LIN {X 0,Y 466.726,Z 1100.087,A -85,B 0,C 180,E1 19216.382,E2 19216.382} C_VEL
LIN {X 0,Y 459.016,Z 1120.699,A -85,B 0,C 180,E1 19214.007,E2 19214.007} C_VEL
LIN {X 0,Y 452.977,Z 1136.346,A -85,B 0,C 180,E1 19211.936,E2 19211.936} C_VEL
LIN {X 0,Y 447.551,Z 1150.209,A -85,B 0,C 180,E1 19209.871,E2 19209.871} C_VEL
LIN {X 0,Y 442.276,Z 1163.7,A -85,B 0,C 180,E1 19207.609,E2 19207.609} C_VEL
LIN {X 0,Y 436.923,Z 1177.533,A -85,B 0,C 180,E1 19204.987,E2 19204.987} C_VEL
LIN {X 0,Y 430.904,Z 1193.503,A -85,B 0,C 180,E1 19201.464,E2 19201.464} C_VEL
LIN {X 0,Y 426.882,Z 1204.833,A -85,B 0,C 180,E1 19198.535,E2 19198.535} C_VEL
LIN {X 0,Y 423.763,Z 1214.343,A -85,B 0,C 180,E1 19195.723,E2 19195.723} C_VEL
LIN {X 0,Y 421.063,Z 1223.466,A -85,B 0,C 180,E1 19192.617,E2 19192.617} C_VEL
LIN {X 0,Y 418.595,Z 1233.141,A -85,B 0,C 180,E1 19188.66,E2 19188.66} C_VEL
LIN {X 0,Y 417.349,Z 1239.293,A -85,B 0,C 180,E1 19185.558,E2 19185.558} C_VEL
LIN {X 0,Y 416.602,Z 1244.084,A -85,B 0,C 180,E1 19182.608,E2 19182.608} C_VEL
LIN {X 0,Y 416.536,Z 1244.656,A -85,B 0,C 180,E1 19182.208,E2 19182.208} C_VEL
LIN {X 0,Y 415.382,Z 1246.217,A -85,B 0,C 180,E1 19181.171,E2 19181.171} C_VEL
LIN {X 0,Y 408.591,Z 1249.799,A -85,B 0,C 180,E1 19178.242,E2 19178.242} C_VEL
LIN {X 0,Y 408.036,Z 1250.419,A -85,B 0,C 180,E1 19177.468,E2 19177.468} C_VEL
LIN {X 0,Y 407.953,Z 1252.387,A -85,B 0,C 180,E1 19174.492,E2 19174.492} C_VEL
LIN {X 0,Y 407.933,Z 1253.358,A -85,B 0,C 180,E1 19171.679,E2 19171.679} C_VEL
LIN {X 0,Y 407.906,Z 1253.459,A -85,B 0,C 180,E1 19168.87,E2 19168.87} C_VEL
LIN {X 0,Y 407.952,Z 1252.658,A -85,B 0,C 180,E1 19165.999,E2 19165.999} C_VEL
LIN {X 0,Y 408.019,Z 1250.929,A -85,B 0,C 180,E1 19163.097,E2 19163.097} C_VEL
LIN {X 0,Y 408.169,Z 1248.351,A -85,B 0,C 180,E1 19160.263,E2 19160.263} C_VEL
LIN {X 0,Y 408.603,Z 1244.86,A -85,B 0,C 180,E1 19157.415,E2 19157.415} C_VEL
LIN {X 0,Y 409.295,Z 1240.436,A -85,B 0,C 180,E1 19154.551,E2 19154.551} C_VEL
LIN {X 0,Y 410.489,Z 1234.748,A -85,B 0,C 180,E1 19151.533,E2 19151.533} C_VEL
LIN {X 0,Y 412.211,Z 1227.955,A -85,B 0,C 180,E1 19148.508,E2 19148.508} C_VEL
LIN {X 0,Y 415.091,Z 1218.417,A -85,B 0,C 180,E1 19144.91,E2 19144.91} C_VEL
LIN {X 0,Y 418.953,Z 1206.868,A -85,B 0,C 180,E1 19141.328,E2 19141.328} C_VEL
LIN {X 0,Y 422.851,Z 1196.299,A -85,B 0,C 180,E1 19138.489,E2 19138.489} C_VEL
LIN {X 0,Y 427.224,Z 1185.009,A -85,B 0,C 180,E1 19135.821,E2 19135.821} C_VEL
LIN {X 0,Y 433.187,Z 1170.311,A -85,B 0,C 180,E1 19132.782,E2 19132.782} C_VEL
LIN {X 0,Y 440.181,Z 1153.04,A -85,B 0,C 180,E1 19129.751,E2 19129.751} C_VEL
LIN {X 0,Y 446.161,Z 1138.346,A -85,B 0,C 180,E1 19127.504,E2 19127.504} C_VEL
LIN {X 0,Y 452.131,Z 1123.44,A -85,B 0,C 180,E1 19125.484,E2 19125.484} C_VEL
LIN {X 0,Y 458.329,Z 1107.59,A -85,B 0,C 180,E1 19123.582,E2 19123.582} C_VEL
LIN {X 0,Y 466.092,Z 1087.076,A -85,B 0,C 180,E1 19121.425,E2 19121.425} C_VEL
LIN {X 0,Y 473.649,Z 1065.436,A -85,B 0,C 180,E1 19119.499,E2 19119.499} C_VEL
LIN {X 0,Y 479.534,Z 1047.568,A -85,B 0,C 180,E1 19118.112,E2 19118.112} C_VEL
LIN {X 0,Y 485.331,Z 1028.607,A -85,B 0,C 180,E1 19116.819,E2 19116.819} C_VEL
LIN {X 0,Y 491.208,Z 1007.732,A -85,B 0,C 180,E1 19115.585,E2 19115.585} C_VEL
LIN {X 0,Y 497.603,Z 982.362,A -85,B 0,C 180,E1 19114.319,E2 19114.319} C_VEL
LIN {X 0,Y 502.722,Z 958.44,A -85,B 0,C 180,E1 19113.342,E2 19113.342} C_VEL
LIN {X 0,Y 506.626,Z 937.283,A -85,B 0,C 180,E1 19112.624,E2 19112.624} C_VEL
LIN {X 0,Y 509.947,Z 915.923,A -85,B 0,C 180,E1 19112.03,E2 19112.03} C_VEL
LIN {X 0,Y 512.846,Z 892.593,A -85,B 0,C 180,E1 19111.515,E2 19111.515} C_VEL
LIN {X 0,Y 515.629,Z 856.761,A -85,B 0,C 180,E1 19110.915,E2 19110.915} C_VEL
LIN {X 0,Y 529.358,Z 635.561,A -85,B 0,C 180,E1 19107.486,E2 19107.486} C_VEL
LIN {X 0,Y 533.456,Z 570.989,A -85,B 0,C 180,E1 19106.464,E2 19106.464} C_VEL
LIN {X 0,Y 524.737,Z 558.021,A -85,B 0,C 180,E1 19104.036,E2 19104.036} C_VEL
LIN {X 0,Y 516.788,Z 546.823,A -85,B 0,C 180,E1 19101.539,E2 19101.539} C_VEL
LIN {X 0,Y 510.867,Z 538.783,A -85,B 0,C 180,E1 19099.435,E2 19099.435} C_VEL
LIN {X 0,Y 506.895,Z 533.497,A -85,B 0,C 180,E1 19097.863,E2 19097.863} C_VEL
LIN {X 0,Y 503.376,Z 528.832,A -85,B 0,C 180,E1 19096.324,E2 19096.324} C_VEL
LIN {X 0,Y 499.419,Z 523.648,A -85,B 0,C 180,E1 19094.375,E2 19094.375} C_VEL
LIN {X 0,Y 496.052,Z 519.314,A -85,B 0,C 180,E1 19092.455,E2 19092.455} C_VEL
LIN {X 0,Y 495.152,Z 518.176,A -85,B 0,C 180,E1 19091.887,E2 19091.887} C_VEL
LIN {X 0,Y 491.947,Z 514.441,A -85,B 0,C 180,E1 19089.594,E2 19089.594} C_VEL
LIN {X 0,Y 490.94,Z 512.514,A -85,B 0,C 180,E1 19088.668,E2 19088.668} C_VEL
LIN {X 0,Y 487.515,Z 509.124,A -85,B 0,C 180,E1 19084.706,E2 19084.706} C_VEL
LIN {X 0,Y 486.689,Z 506.403,A -85,B 0,C 180,E1 19082.355,E2 19082.355} C_VEL
LIN {X 0,Y 486.775,Z 506.534,A -85,B 0,C 180,E1 19077.763,E2 19077.763} C_VEL
LIN {X 0,Y 488.567,Z 510.725,A -85,B 0,C 180,E1 19074.127,E2 19074.127} C_VEL
LIN {X 0,Y 491.202,Z 512.848,A -85,B 0,C 180,E1 19071.513,E2 19071.513} C_VEL
LIN {X 0,Y 493.665,Z 516.868,A -85,B 0,C 180,E1 19069.497,E2 19069.497} C_VEL
LIN {X 0,Y 495.884,Z 519.004,A -85,B 0,C 180,E1 19068.072,E2 19068.072} C_VEL
LIN {X 0,Y 499.313,Z 523.558,A -85,B 0,C 180,E1 19066.095,E2 19066.095} C_VEL
LIN {X 0,Y 500.82,Z 525.628,A -85,B 0,C 180,E1 19065.312,E2 19065.312} C_VEL
LIN {X 0,Y 505.099,Z 531.129,A -85,B 0,C 180,E1 19063.319,E2 19063.319} C_VEL
LIN {X 0,Y 511.053,Z 540.056,A -85,B 0,C 180,E1 19060.87,E2 19060.87} C_VEL
LIN {X 0,Y 516.454,Z 548.16,A -85,B 0,C 180,E1 19058.923,E2 19058.923} C_VEL
LIN {X 0,Y 524.596,Z 561.043,A -85,B 0,C 180,E1 19056.316,E2 19056.316} C_VEL
LIN {X 0,Y 533.578,Z 575.978,A -85,B 0,C 180,E1 19053.779,E2 19053.779} C_VEL
LIN {X 0,Y 520.443,Z 784.729,A -85,B 0,C 180,E1 19050.532,E2 19050.532} C_VEL
LIN {X 0,Y 513.397,Z 898.299,A -85,B 0,C 180,E1 19048.753,E2 19048.753} C_VEL
LIN {X 0,Y 510.438,Z 925.967,A -85,B 0,C 180,E1 19048.226,E2 19048.226} C_VEL
LIN {X 0,Y 506.32,Z 952.366,A -85,B 0,C 180,E1 19047.555,E2 19047.555} C_VEL
LIN {X 0,Y 502.372,Z 973.666,A -85,B 0,C 180,E1 19046.874,E2 19046.874} C_VEL
LIN {X 0,Y 497.981,Z 994.234,A -85,B 0,C 180,E1 19046.088,E2 19046.088} C_VEL
LIN {X 0,Y 492.921,Z 1015.345,A -85,B 0,C 180,E1 19045.132,E2 19045.132} C_VEL
LIN {X 0,Y 486.06,Z 1040.963,A -85,B 0,C 180,E1 19043.75,E2 19043.75} C_VEL
LIN {X 0,Y 479.409,Z 1062.995,A -85,B 0,C 180,E1 19042.331,E2 19042.331} C_VEL
LIN {X 0,Y 473.078,Z 1082.578,A -85,B 0,C 180,E1 19040.872,E2 19040.872} C_VEL
LIN {X 0,Y 466.468,Z 1101.878,A -85,B 0,C 180,E1 19039.224,E2 19039.224} C_VEL
LIN {X 0,Y 458.48,Z 1124.086,A -85,B 0,C 180,E1 19037.033,E2 19037.033} C_VEL
LIN {X 0,Y 450.994,Z 1143.777,A -85,B 0,C 180,E1 19034.747,E2 19034.747} C_VEL
LIN {X 0,Y 445.06,Z 1159.134,A -85,B 0,C 180,E1 19032.722,E2 19032.722} C_VEL
LIN {X 0,Y 439.157,Z 1174.316,A -85,B 0,C 180,E1 19030.464,E2 19030.464} C_VEL
LIN {X 0,Y 432.558,Z 1191.551,A -85,B 0,C 180,E1 19027.545,E2 19027.545} C_VEL
LIN {X 0,Y 426.449,Z 1207.49,A -85,B 0,C 180,E1 19024.378,E2 19024.378} C_VEL
LIN {X 0,Y 421.982,Z 1219.772,A -85,B 0,C 180,E1 19021.583,E2 19021.583} C_VEL
LIN {X 0,Y 418.242,Z 1230.826,A -85,B 0,C 180,E1 19018.725,E2 19018.725} C_VEL
LIN {X 0,Y 414.529,Z 1242.95,A -85,B 0,C 180,E1 19015.126,E2 19015.126} C_VEL
LIN {X 0,Y 411.805,Z 1253.015,A -85,B 0,C 180,E1 19011.514,E2 19011.514} C_VEL
LIN {X 0,Y 410.172,Z 1260.206,A -85,B 0,C 180,E1 19008.481,E2 19008.481} C_VEL
LIN {X 0,Y 409.136,Z 1265.988,A -85,B 0,C 180,E1 19005.6,E2 19005.6} C_VEL
LIN {X 0,Y 408.459,Z 1270.971,A -85,B 0,C 180,E1 19002.59,E2 19002.59} C_VEL
LIN {X 0,Y 408.085,Z 1274.707,A -85,B 0,C 180,E1 18999.739,E2 18999.739} C_VEL
LIN {X 0,Y 407.978,Z 1277.483,A -85,B 0,C 180,E1 18996.903,E2 18996.903} C_VEL
LIN {X 0,Y 407.935,Z 1279.311,A -85,B 0,C 180,E1 18994.082,E2 18994.082} C_VEL
LIN {X 0,Y 407.921,Z 1280.177,A -85,B 0,C 180,E1 18991.411,E2 18991.411} C_VEL
LIN {X 0,Y 407.915,Z 1280.202,A -85,B 0,C 180,E1 18988.742,E2 18988.742} C_VEL
LIN {X 0,Y 407.935,Z 1279.368,A -85,B 0,C 180,E1 18986.032,E2 18986.032} C_VEL
LIN {X 0,Y 407.973,Z 1277.61,A -85,B 0,C 180,E1 18983.251,E2 18983.251} C_VEL
LIN {X 0,Y 408.073,Z 1274.886,A -85,B 0,C 180,E1 18980.416,E2 18980.416} C_VEL
LIN {X 0,Y 408.435,Z 1271.203,A -85,B 0,C 180,E1 18977.566,E2 18977.566} C_VEL
LIN {X 0,Y 409.082,Z 1266.273,A -85,B 0,C 180,E1 18974.556,E2 18974.556} C_VEL
LIN {X 0,Y 410.105,Z 1260.544,A -85,B 0,C 180,E1 18971.676,E2 18971.676} C_VEL
LIN {X 0,Y 411.701,Z 1253.406,A -85,B 0,C 180,E1 18968.644,E2 18968.644} C_VEL
LIN {X 0,Y 414.263,Z 1243.805,A -85,B 0,C 180,E1 18965.168,E2 18965.168} C_VEL
LIN {X 0,Y 418.052,Z 1231.399,A -85,B 0,C 180,E1 18961.431,E2 18961.431} C_VEL
LIN {X 0,Y 421.762,Z 1220.406,A -85,B 0,C 180,E1 18958.572,E2 18958.572} C_VEL
LIN {X 0,Y 425.986,Z 1208.695,A -85,B 0,C 180,E1 18955.885,E2 18955.885} C_VEL
LIN {X 0,Y 431.201,Z 1194.919,A -85,B 0,C 180,E1 18953.099,E2 18953.099} C_VEL
LIN {X 0,Y 438.495,Z 1176.02,A -85,B 0,C 180,E1 18949.809,E2 18949.809} C_VEL
LIN {X 0,Y 444.678,Z 1160.077,A -85,B 0,C 180,E1 18947.416,E2 18947.416} C_VEL
LIN {X 0,Y 450.753,Z 1144.339,A -85,B 0,C 180,E1 18945.328,E2 18945.328} C_VEL
LIN {X 0,Y 457.565,Z 1126.379,A -85,B 0,C 180,E1 18943.228,E2 18943.228} C_VEL
LIN {X 0,Y 466.103,Z 1102.816,A -85,B 0,C 180,E1 18940.866,E2 18940.866} C_VEL
LIN {X 0,Y 472.749,Z 1083.429,A -85,B 0,C 180,E1 18939.202,E2 18939.202} C_VEL
LIN {X 0,Y 478.837,Z 1064.661,A -85,B 0,C 180,E1 18937.793,E2 18937.793} C_VEL
LIN {X 0,Y 484.915,Z 1044.638,A -85,B 0,C 180,E1 18936.483,E2 18936.483} C_VEL
LIN {X 0,Y 491.767,Z 1019.829,A -85,B 0,C 180,E1 18935.09,E2 18935.09} C_VEL
LIN {X 0,Y 497.452,Z 996.33,A -85,B 0,C 180,E1 18934.005,E2 18934.005} C_VEL
LIN {X 0,Y 502.002,Z 975.19,A -85,B 0,C 180,E1 18933.184,E2 18933.184} C_VEL
LIN {X 0,Y 505.927,Z 954.249,A -85,B 0,C 180,E1 18932.506,E2 18932.506} C_VEL
LIN {X 0,Y 509.434,Z 932.151,A -85,B 0,C 180,E1 18931.924,E2 18931.924} C_VEL
LIN {X 0,Y 512.865,Z 904.139,A -85,B 0,C 180,E1 18931.35,E2 18931.35} C_VEL
LIN {X 0,Y 515.951,Z 857.879,A -85,B 0,C 180,E1 18930.607,E2 18930.607} C_VEL
LIN {X 0,Y 529.334,Z 640.596,A -85,B 0,C 180,E1 18927.234,E2 18927.234} C_VEL
LIN {X 0,Y 533.472,Z 575.938,A -85,B 0,C 180,E1 18926.223,E2 18926.223} C_VEL
LIN {X 0,Y 524.4,Z 560.859,A -85,B 0,C 180,E1 18923.664,E2 18923.664} C_VEL
LIN {X 0,Y 516.019,Z 547.617,A -85,B 0,C 180,E1 18920.977,E2 18920.977} C_VEL
LIN {X 0,Y 509.259,Z 537.343,A -85,B 0,C 180,E1 18918.487,E2 18918.487} C_VEL
LIN {X 0,Y 503.589,Z 529.163,A -85,B 0,C 180,E1 18916.08,E2 18916.08} C_VEL
LIN {X 0,Y 499.246,Z 523.57,A -85,B 0,C 180,E1 18913.966,E2 18913.966} C_VEL
LIN {X 0,Y 495.613,Z 518.693,A -85,B 0,C 180,E1 18911.875,E2 18911.875} C_VEL
LIN {X 0,Y 492.093,Z 514.875,A -85,B 0,C 180,E1 18909.473,E2 18909.473} C_VEL
LIN {X 0,Y 490.793,Z 512.489,A -85,B 0,C 180,E1 18908.317,E2 18908.317} C_VEL
LIN {X 0,Y 487.383,Z 509.118,A -85,B 0,C 180,E1 18904.471,E2 18904.471} C_VEL
LIN {X 0,Y 486.52,Z 506.4,A -85,B 0,C 180,E1 18902.238,E2 18902.238} C_VEL
LIN {X 0,Y 486.665,Z 506.642,A -85,B 0,C 180,E1 18896.82,E2 18896.82} C_VEL
LIN {X 0,Y 487.967,Z 510.023,A -85,B 0,C 180,E1 18894.119,E2 18894.119} C_VEL
LIN {X 0,Y 491.082,Z 512.857,A -85,B 0,C 180,E1 18890.921,E2 18890.921} C_VEL
LIN {X 0,Y 493.424,Z 516.662,A -85,B 0,C 180,E1 18889.019,E2 18889.019} C_VEL
LIN {X 0,Y 495.739,Z 518.901,A -85,B 0,C 180,E1 18887.537,E2 18887.537} C_VEL
LIN {X 0,Y 499.073,Z 523.419,A -85,B 0,C 180,E1 18885.615,E2 18885.615} C_VEL
LIN {X 0,Y 500.379,Z 525.041,A -85,B 0,C 180,E1 18884.943,E2 18884.943} C_VEL
LIN {X 0,Y 504.758,Z 530.701,A -85,B 0,C 180,E1 18882.892,E2 18882.892} C_VEL
LIN {X 0,Y 508.971,Z 536.338,A -85,B 0,C 180,E1 18881.145,E2 18881.145} C_VEL
LIN {X 0,Y 513.583,Z 542.55,A -85,B 0,C 180,E1 18879.426,E2 18879.426} C_VEL
LIN {X 0,Y 519.796,Z 551.145,A -85,B 0,C 180,E1 18877.343,E2 18877.343} C_VEL
LIN {X 0,Y 526.736,Z 561.091,A -85,B 0,C 180,E1 18875.255,E2 18875.255} C_VEL
LIN {X 0,Y 533.433,Z 571.162,A -85,B 0,C 180,E1 18873.42,E2 18873.42} C_VEL
LIN {X 0,Y 519.648,Z 789.072,A -85,B 0,C 180,E1 18870.039,E2 18870.039} C_VEL
LIN {X 0,Y 513.854,Z 881.148,A -85,B 0,C 180,E1 18868.594,E2 18868.594} C_VEL
LIN {X 0,Y 510.941,Z 908.605,A -85,B 0,C 180,E1 18868.056,E2 18868.056} C_VEL
LIN {X 0,Y 507.028,Z 934.536,A -85,B 0,C 180,E1 18867.364,E2 18867.364} C_VEL
LIN {X 0,Y 503.185,Z 955.72,A -85,B 0,C 180,E1 18866.662,E2 18866.662} C_VEL
LIN {X 0,Y 498.898,Z 976.164,A -85,B 0,C 180,E1 18865.852,E2 18865.852} C_VEL
LIN {X 0,Y 493.586,Z 998.455,A -85,B 0,C 180,E1 18864.811,E2 18864.811} C_VEL
LIN {X 0,Y 486.295,Z 1025.23,A -85,B 0,C 180,E1 18863.298,E2 18863.298} C_VEL
LIN {X 0,Y 480.324,Z 1044.924,A -85,B 0,C 180,E1 18861.982,E2 18861.982} C_VEL
LIN {X 0,Y 474.546,Z 1062.594,A -85,B 0,C 180,E1 18860.637,E2 18860.637} C_VEL
LIN {X 0,Y 468.3,Z 1080.543,A -85,B 0,C 180,E1 18859.087,E2 18859.087} C_VEL
LIN {X 0,Y 461.069,Z 1100.356,A -85,B 0,C 180,E1 18857.126,E2 18857.126} C_VEL
LIN {X 0,Y 452.98,Z 1121.24,A -85,B 0,C 180,E1 18854.702,E2 18854.702} C_VEL
LIN {X 0,Y 446.89,Z 1136.46,A -85,B 0,C 180,E1 18852.672,E2 18852.672} C_VEL
LIN {X 0,Y 441.191,Z 1150.486,A -85,B 0,C 180,E1 18850.564,E2 18850.564} C_VEL
LIN {X 0,Y 435.693,Z 1163.977,A -85,B 0,C 180,E1 18848.279,E2 18848.279} C_VEL
LIN {X 0,Y 430.208,Z 1177.547,A -85,B 0,C 180,E1 18845.678,E2 18845.678} C_VEL
LIN {X 0,Y 423.945,Z 1193.42,A -85,B 0,C 180,E1 18842.143,E2 18842.143} C_VEL
LIN {X 0,Y 419.776,Z 1204.605,A -85,B 0,C 180,E1 18839.22,E2 18839.22} C_VEL
LIN {X 0,Y 416.446,Z 1214.17,A -85,B 0,C 180,E1 18836.363,E2 18836.363} C_VEL
LIN {X 0,Y 413.649,Z 1222.95,A -85,B 0,C 180,E1 18833.347,E2 18833.347} C_VEL
LIN {X 0,Y 411.21,Z 1231.897,A -85,B 0,C 180,E1 18829.746,E2 18829.746} C_VEL
LIN {X 0,Y 409.539,Z 1239.316,A -85,B 0,C 180,E1 18826.007,E2 18826.007} C_VEL
LIN {X 0,Y 408.666,Z 1244.352,A -85,B 0,C 180,E1 18822.857,E2 18822.857} C_VEL
LIN {X 0,Y 408.212,Z 1247.956,A -85,B 0,C 180,E1 18820.008,E2 18820.008} C_VEL
LIN {X 0,Y 408.036,Z 1250.419,A -85,B 0,C 180,E1 18817.468,E2 18817.468} C_VEL
LIN {X 0,Y 407.031,Z 1251.303,A -85,B 0,C 180,E1 18816.394,E2 18816.394} C_VEL
LIN {X 0,Y 402.53,Z 1252.744,A -85,B 0,C 180,E1 18814.442,E2 18814.442} C_VEL
LIN {X 0,Y 400.152,Z 1253.388,A -85,B 0,C 180,E1 18813.044,E2 18813.044} C_VEL
LIN {X 0,Y 399.942,Z 1253.493,A -85,B 0,C 180,E1 18812.565,E2 18812.565} C_VEL
LIN {X 0,Y 399.899,Z 1253.766,A -85,B 0,C 180,E1 18809.134,E2 18809.134} C_VEL
LIN {X 0,Y 399.956,Z 1253.015,A -85,B 0,C 180,E1 18806.123,E2 18806.123} C_VEL
LIN {X 0,Y 400.027,Z 1251.303,A -85,B 0,C 180,E1 18803.103,E2 18803.103} C_VEL
LIN {X 0,Y 400.187,Z 1248.77,A -85,B 0,C 180,E1 18800.212,E2 18800.212} C_VEL
LIN {X 0,Y 400.639,Z 1245.326,A -85,B 0,C 180,E1 18797.307,E2 18797.307} C_VEL
LIN {X 0,Y 401.428,Z 1240.703,A -85,B 0,C 180,E1 18794.241,E2 18794.241} C_VEL
LIN {X 0,Y 402.693,Z 1235.017,A -85,B 0,C 180,E1 18791.163,E2 18791.163} C_VEL
LIN {X 0,Y 404.669,Z 1227.823,A -85,B 0,C 180,E1 18787.909,E2 18787.909} C_VEL
LIN {X 0,Y 408.024,Z 1217.356,A -85,B 0,C 180,E1 18783.977,E2 18783.977} C_VEL
LIN {X 0,Y 411.858,Z 1206.636,A -85,B 0,C 180,E1 18780.627,E2 18780.627} C_VEL
LIN {X 0,Y 415.966,Z 1196.01,A -85,B 0,C 180,E1 18777.743,E2 18777.743} C_VEL
LIN {X 0,Y 420.869,Z 1184.036,A -85,B 0,C 180,E1 18774.9,E2 18774.9} C_VEL
LIN {X 0,Y 428.108,Z 1166.888,A -85,B 0,C 180,E1 18771.415,E2 18771.415} C_VEL
LIN {X 0,Y 434.058,Z 1152.818,A -85,B 0,C 180,E1 18768.96,E2 18768.96} C_VEL
LIN {X 0,Y 440.286,Z 1138.072,A -85,B 0,C 180,E1 18766.693,E2 18766.693} C_VEL
LIN {X 0,Y 446.663,Z 1122.709,A -85,B 0,C 180,E1 18764.608,E2 18764.608} C_VEL
LIN {X 0,Y 454.218,Z 1104.044,A -85,B 0,C 180,E1 18762.387,E2 18762.387} C_VEL
LIN {X 0,Y 462.554,Z 1082.074,A -85,B 0,C 180,E1 18760.164,E2 18760.164} C_VEL
LIN {X 0,Y 469.222,Z 1063.518,A -85,B 0,C 180,E1 18758.546,E2 18758.546} C_VEL
LIN {X 0,Y 475.159,Z 1045.929,A -85,B 0,C 180,E1 18757.199,E2 18757.199} C_VEL
LIN {X 0,Y 481.024,Z 1027.163,A -85,B 0,C 180,E1 18755.935,E2 18755.935} C_VEL
LIN {X 0,Y 487.958,Z 1003,A -85,B 0,C 180,E1 18754.534,E2 18754.534} C_VEL
LIN {X 0,Y 494.079,Z 978.214,A -85,B 0,C 180,E1 18753.354,E2 18753.354} C_VEL
LIN {X 0,Y 498.516,Z 957.806,A -85,B 0,C 180,E1 18752.536,E2 18752.536} C_VEL
LIN {X 0,Y 502.448,Z 936.913,A -85,B 0,C 180,E1 18751.833,E2 18751.833} C_VEL
LIN {X 0,Y 505.871,Z 915.263,A -85,B 0,C 180,E1 18751.237,E2 18751.237} C_VEL
LIN {X 0,Y 509.187,Z 888.849,A -85,B 0,C 180,E1 18750.668,E2 18750.668} C_VEL
LIN {X 0,Y 512.187,Z 846.85,A -85,B 0,C 180,E1 18749.988,E2 18749.988} C_VEL
LIN {X 0,Y 526.264,Z 627.318,A -85,B 0,C 180,E1 18746.578,E2 18746.578} C_VEL
LIN {X 0,Y 529.65,Z 575.892,A -85,B 0,C 180,E1 18745.768,E2 18745.768} C_VEL
LIN {X 0,Y 521.588,Z 563.831,A -85,B 0,C 180,E1 18743.44,E2 18743.44} C_VEL
LIN {X 0,Y 513.424,Z 552.013,A -85,B 0,C 180,E1 18740.76,E2 18740.76} C_VEL
LIN {X 0,Y 505.79,Z 541.654,A -85,B 0,C 180,E1 18737.844,E2 18737.844} C_VEL
LIN {X 0,Y 501.796,Z 536.391,A -85,B 0,C 180,E1 18736.08,E2 18736.08} C_VEL
LIN {X 0,Y 497.908,Z 531.249,A -85,B 0,C 180,E1 18734.123,E2 18734.123} C_VEL
LIN {X 0,Y 494.538,Z 526.701,A -85,B 0,C 180,E1 18732.139,E2 18732.139} C_VEL
LIN {X 0,Y 490.628,Z 522.009,A -85,B 0,C 180,E1 18729.324,E2 18729.324} C_VEL
LIN {X 0,Y 489.699,Z 520.334,A -85,B 0,C 180,E1 18728.454,E2 18728.454} C_VEL
LIN {X 0,Y 486.356,Z 516.74,A -85,B 0,C 180,E1 18724.363,E2 18724.363} C_VEL
LIN {X 0,Y 485.679,Z 514.337,A -85,B 0,C 180,E1 18722.242,E2 18722.242} C_VEL
LIN {X 0,Y 485.788,Z 514.581,A -85,B 0,C 180,E1 18717.759,E2 18717.759} C_VEL
LIN {X 0,Y 487.592,Z 518.707,A -85,B 0,C 180,E1 18714.115,E2 18714.115} C_VEL
LIN {X 0,Y 490.084,Z 520.819,A -85,B 0,C 180,E1 18711.612,E2 18711.612} C_VEL
LIN {X 0,Y 492.692,Z 524.929,A -85,B 0,C 180,E1 18709.476,E2 18709.476} C_VEL
LIN {X 0,Y 494.626,Z 526.862,A -85,B 0,C 180,E1 18708.219,E2 18708.219} C_VEL
LIN {X 0,Y 498.128,Z 531.455,A -85,B 0,C 180,E1 18706.18,E2 18706.18} C_VEL
LIN {X 0,Y 503.735,Z 539.035,A -85,B 0,C 180,E1 18703.451,E2 18703.451} C_VEL
LIN {X 0,Y 510.055,Z 548.657,A -85,B 0,C 180,E1 18700.831,E2 18700.831} C_VEL
LIN {X 0,Y 516.373,Z 558.466,A -85,B 0,C 180,E1 18698.562,E2 18698.562} C_VEL
LIN {X 0,Y 524.604,Z 571.867,A -85,B 0,C 180,E1 18695.958,E2 18695.958} C_VEL
LIN {X 0,Y 529.731,Z 580.871,A -85,B 0,C 180,E1 18694.478,E2 18694.478} C_VEL
LIN {X 0,Y 515.713,Z 797.428,A -85,B 0,C 180,E1 18691.109,E2 18691.109} C_VEL
LIN {X 0,Y 509.25,Z 898.269,A -85,B 0,C 180,E1 18689.524,E2 18689.524} C_VEL
LIN {X 0,Y 506.182,Z 926.092,A -85,B 0,C 180,E1 18688.993,E2 18688.993} C_VEL
LIN {X 0,Y 502.01,Z 952.22,A -85,B 0,C 180,E1 18688.33,E2 18688.33} C_VEL
LIN {X 0,Y 497.985,Z 973.408,A -85,B 0,C 180,E1 18687.656,E2 18687.656} C_VEL
LIN {X 0,Y 493.607,Z 993.448,A -85,B 0,C 180,E1 18686.894,E2 18686.894} C_VEL
LIN {X 0,Y 488.609,Z 1013.832,A -85,B 0,C 180,E1 18685.979,E2 18685.979} C_VEL
LIN {X 0,Y 482.072,Z 1037.87,A -85,B 0,C 180,E1 18684.709,E2 18684.709} C_VEL
LIN {X 0,Y 474.674,Z 1061.901,A -85,B 0,C 180,E1 18683.179,E2 18683.179} C_VEL
LIN {X 0,Y 468.217,Z 1081.365,A -85,B 0,C 180,E1 18681.735,E2 18681.735} C_VEL
LIN {X 0,Y 461.927,Z 1099.258,A -85,B 0,C 180,E1 18680.218,E2 18680.218} C_VEL
LIN {X 0,Y 455.316,Z 1117.16,A -85,B 0,C 180,E1 18678.495,E2 18678.495} C_VEL
LIN {X 0,Y 447.394,Z 1137.849,A -85,B 0,C 180,E1 18676.215,E2 18676.215} C_VEL
LIN {X 0,Y 439.422,Z 1157.591,A -85,B 0,C 180,E1 18673.647,E2 18673.647} C_VEL
LIN {X 0,Y 433.347,Z 1172.593,A -85,B 0,C 180,E1 18671.419,E2 18671.419} C_VEL
LIN {X 0,Y 427.502,Z 1187.038,A -85,B 0,C 180,E1 18668.994,E2 18668.994} C_VEL
LIN {X 0,Y 421.138,Z 1203.157,A -85,B 0,C 180,E1 18665.91,E2 18665.91} C_VEL
LIN {X 0,Y 415.448,Z 1217.814,A -85,B 0,C 180,E1 18662.608,E2 18662.608} C_VEL
LIN {X 0,Y 411.416,Z 1228.972,A -85,B 0,C 180,E1 18659.727,E2 18659.727} C_VEL
LIN {X 0,Y 408.093,Z 1238.923,A -85,B 0,C 180,E1 18656.802,E2 18656.802} C_VEL
LIN {X 0,Y 405.319,Z 1248.088,A -85,B 0,C 180,E1 18653.716,E2 18653.716} C_VEL
LIN {X 0,Y 402.821,Z 1257.89,A -85,B 0,C 180,E1 18649.819,E2 18649.819} C_VEL
LIN {X 0,Y 401.333,Z 1265.195,A -85,B 0,C 180,E1 18646.209,E2 18646.209} C_VEL
LIN {X 0,Y 400.551,Z 1270.277,A -85,B 0,C 180,E1 18643.136,E2 18643.136} C_VEL
LIN {X 0,Y 400.141,Z 1274.111,A -85,B 0,C 180,E1 18640.225,E2 18640.225} C_VEL
LIN {X 0,Y 399.989,Z 1276.984,A -85,B 0,C 180,E1 18637.331,E2 18637.331} C_VEL
LIN {X 0,Y 399.939,Z 1278.907,A -85,B 0,C 180,E1 18634.451,E2 18634.451} C_VEL
LIN {X 0,Y 399.933,Z 1279.868,A -85,B 0,C 180,E1 18631.726,E2 18631.726} C_VEL
LIN {X 0,Y 399.904,Z 1279.986,A -85,B 0,C 180,E1 18629.004,E2 18629.004} C_VEL
LIN {X 0,Y 399.937,Z 1279.194,A -85,B 0,C 180,E1 18626.136,E2 18626.136} C_VEL
LIN {X 0,Y 399.974,Z 1277.463,A -85,B 0,C 180,E1 18623.259,E2 18623.259} C_VEL
LIN {X 0,Y 400.076,Z 1274.785,A -85,B 0,C 180,E1 18620.368,E2 18620.368} C_VEL
LIN {X 0,Y 400.471,Z 1270.935,A -85,B 0,C 180,E1 18617.315,E2 18617.315} C_VEL
LIN {X 0,Y 401.183,Z 1266.003,A -85,B 0,C 180,E1 18614.244,E2 18614.244} C_VEL
LIN {X 0,Y 402.279,Z 1260.182,A -85,B 0,C 180,E1 18611.263,E2 18611.263} C_VEL
LIN {X 0,Y 404.064,Z 1252.77,A -85,B 0,C 180,E1 18608.067,E2 18608.067} C_VEL
LIN {X 0,Y 407.084,Z 1242.25,A -85,B 0,C 180,E1 18604.239,E2 18604.239} C_VEL
LIN {X 0,Y 410.865,Z 1230.596,A -85,B 0,C 180,E1 18600.724,E2 18600.724} C_VEL
LIN {X 0,Y 414.571,Z 1220.127,A -85,B 0,C 180,E1 18597.963,E2 18597.963} C_VEL
LIN {X 0,Y 419.015,Z 1208.416,A -85,B 0,C 180,E1 18595.237,E2 18595.237} C_VEL
LIN {X 0,Y 424.478,Z 1194.64,A -85,B 0,C 180,E1 18592.414,E2 18592.414} C_VEL
LIN {X 0,Y 432.045,Z 1175.801,A -85,B 0,C 180,E1 18589.095,E2 18589.095} C_VEL
LIN {X 0,Y 438.506,Z 1159.79,A -85,B 0,C 180,E1 18586.668,E2 18586.668} C_VEL
LIN {X 0,Y 444.807,Z 1144.06,A -85,B 0,C 180,E1 18584.566,E2 18584.566} C_VEL
LIN {X 0,Y 452.087,Z 1125.538,A -85,B 0,C 180,E1 18582.39,E2 18582.39} C_VEL
LIN {X 0,Y 460.692,Z 1102.555,A -85,B 0,C 180,E1 18580.084,E2 18580.084} C_VEL
LIN {X 0,Y 467.573,Z 1083.079,A -85,B 0,C 180,E1 18578.408,E2 18578.408} C_VEL
LIN {X 0,Y 474.076,Z 1063.567,A -85,B 0,C 180,E1 18576.945,E2 18576.945} C_VEL
LIN {X 0,Y 480.894,Z 1041.641,A -85,B 0,C 180,E1 18575.524,E2 18575.524} C_VEL
LIN {X 0,Y 487.966,Z 1016.14,A -85,B 0,C 180,E1 18574.138,E2 18574.138} C_VEL
LIN {X 0,Y 493.238,Z 994.764,A -85,B 0,C 180,E1 18573.166,E2 18573.166} C_VEL
LIN {X 0,Y 497.759,Z 974.172,A -85,B 0,C 180,E1 18572.376,E2 18572.376} C_VEL
LIN {X 0,Y 501.798,Z 953.002,A -85,B 0,C 180,E1 18571.698,E2 18571.698} C_VEL
LIN {X 0,Y 505.598,Z 929.404,A -85,B 0,C 180,E1 18571.09,E2 18571.09} C_VEL
LIN {X 0,Y 509.051,Z 899.773,A -85,B 0,C 180,E1 18570.507,E2 18570.507} C_VEL
LIN {X 0,Y 513.37,Z 833.721,A -85,B 0,C 180,E1 18569.461,E2 18569.461} C_VEL
LIN {X 0,Y 527.141,Z 618.296,A -85,B 0,C 180,E1 18566.11,E2 18566.11} C_VEL
LIN {X 0,Y 529.557,Z 580.498,A -85,B 0,C 180,E1 18565.5,E2 18565.5} C_VEL
LIN {X 0,Y 521.347,Z 566.607,A -85,B 0,C 180,E1 18563.092,E2 18563.092} C_VEL
LIN {X 0,Y 513.122,Z 553.408,A -85,B 0,C 180,E1 18560.355,E2 18560.355} C_VEL
LIN {X 0,Y 506.364,Z 543.237,A -85,B 0,C 180,E1 18557.763,E2 18557.763} C_VEL
LIN {X 0,Y 501.998,Z 536.726,A -85,B 0,C 180,E1 18555.836,E2 18555.836} C_VEL
LIN {X 0,Y 497.732,Z 531.161,A -85,B 0,C 180,E1 18553.712,E2 18553.712} C_VEL
LIN {X 0,Y 493.901,Z 526.07,A -85,B 0,C 180,E1 18551.443,E2 18551.443} C_VEL
LIN {X 0,Y 490.827,Z 522.564,A -85,B 0,C 180,E1 18549.261,E2 18549.261} C_VEL
LIN {X 0,Y 489.686,Z 520.38,A -85,B 0,C 180,E1 18548.218,E2 18548.218} C_VEL
LIN {X 0,Y 486.337,Z 516.997,A -85,B 0,C 180,E1 18544.363,E2 18544.363} C_VEL
LIN {X 0,Y 485.546,Z 514.34,A -85,B 0,C 180,E1 18542.242,E2 18542.242} C_VEL
LIN {X 0,Y 485.655,Z 514.564,A -85,B 0,C 180,E1 18536.906,E2 18536.906} C_VEL
LIN {X 0,Y 486.907,Z 517.903,A -85,B 0,C 180,E1 18534.225,E2 18534.225} C_VEL
LIN {X 0,Y 489.904,Z 520.693,A -85,B 0,C 180,E1 18531.076,E2 18531.076} C_VEL
LIN {X 0,Y 492.452,Z 524.727,A -85,B 0,C 180,E1 18528.997,E2 18528.997} C_VEL
LIN {X 0,Y 494.395,Z 526.609,A -85,B 0,C 180,E1 18527.739,E2 18527.739} C_VEL
LIN {X 0,Y 497.781,Z 531.22,A -85,B 0,C 180,E1 18525.755,E2 18525.755} C_VEL
LIN {X 0,Y 503.151,Z 538.252,A -85,B 0,C 180,E1 18523.134,E2 18523.134} C_VEL
LIN {X 0,Y 507.165,Z 543.7,A -85,B 0,C 180,E1 18521.434,E2 18521.434} C_VEL
LIN {X 0,Y 513.515,Z 552.297,A -85,B 0,C 180,E1 18519.065,E2 18519.065} C_VEL
LIN {X 0,Y 522.855,Z 565.677,A -85,B 0,C 180,E1 18516.052,E2 18516.052} C_VEL
LIN {X 0,Y 529.587,Z 576.029,A -85,B 0,C 180,E1 18514.124,E2 18514.124} C_VEL
LIN {X 0,Y 515.482,Z 792.776,A -85,B 0,C 180,E1 18510.757,E2 18510.757} C_VEL
LIN {X 0,Y 509.724,Z 881.469,A -85,B 0,C 180,E1 18509.362,E2 18509.362} C_VEL
LIN {X 0,Y 506.727,Z 909.013,A -85,B 0,C 180,E1 18508.822,E2 18508.822} C_VEL
LIN {X 0,Y 502.743,Z 934.812,A -85,B 0,C 180,E1 18508.135,E2 18508.135} C_VEL
LIN {X 0,Y 498.805,Z 955.994,A -85,B 0,C 180,E1 18507.435,E2 18507.435} C_VEL
LIN {X 0,Y 494.414,Z 976.438,A -85,B 0,C 180,E1 18506.626,E2 18506.626} C_VEL
LIN {X 0,Y 488.963,Z 998.728,A -85,B 0,C 180,E1 18505.587,E2 18505.587} C_VEL
LIN {X 0,Y 481.76,Z 1024.611,A -85,B 0,C 180,E1 18504.129,E2 18504.129} C_VEL
LIN {X 0,Y 475.596,Z 1044.419,A -85,B 0,C 180,E1 18502.813,E2 18502.813} C_VEL
LIN {X 0,Y 469.388,Z 1062.868,A -85,B 0,C 180,E1 18501.411,E2 18501.411} C_VEL
LIN {X 0,Y 462.955,Z 1080.818,A -85,B 0,C 180,E1 18499.856,E2 18499.856} C_VEL
LIN {X 0,Y 455.491,Z 1100.631,A -85,B 0,C 180,E1 18497.888,E2 18497.888} C_VEL
LIN {X 0,Y 447.23,Z 1121.251,A -85,B 0,C 180,E1 18495.484,E2 18495.484} C_VEL
LIN {X 0,Y 440.619,Z 1137.193,A -85,B 0,C 180,E1 18493.339,E2 18493.339} C_VEL
LIN {X 0,Y 434.547,Z 1151.594,A -85,B 0,C 180,E1 18491.143,E2 18491.143} C_VEL
LIN {X 0,Y 428.547,Z 1165.768,A -85,B 0,C 180,E1 18488.694,E2 18488.694} C_VEL
LIN {X 0,Y 421.815,Z 1181.866,A -85,B 0,C 180,E1 18485.494,E2 18485.494} C_VEL
LIN {X 0,Y 416.29,Z 1195.178,A -85,B 0,C 180,E1 18482.377,E2 18482.377} C_VEL
LIN {X 0,Y 412.137,Z 1205.887,A -85,B 0,C 180,E1 18479.496,E2 18479.496} C_VEL
LIN {X 0,Y 408.701,Z 1215.34,A -85,B 0,C 180,E1 18476.588,E2 18476.588} C_VEL
LIN {X 0,Y 405.474,Z 1225.197,A -85,B 0,C 180,E1 18473.076,E2 18473.076} C_VEL
LIN {X 0,Y 402.88,Z 1234.273,A -85,B 0,C 180,E1 18469.115,E2 18469.115} C_VEL
LIN {X 0,Y 401.564,Z 1240.099,A -85,B 0,C 180,E1 18466.025,E2 18466.025} C_VEL
LIN {X 0,Y 400.706,Z 1244.82,A -85,B 0,C 180,E1 18462.971,E2 18462.971} C_VEL
LIN {X 0,Y 400.23,Z 1248.376,A -85,B 0,C 180,E1 18460.064,E2 18460.064} C_VEL
LIN {X 0,Y 400.042,Z 1251.022,A -85,B 0,C 180,E1 18457.172,E2 18457.172} C_VEL
LIN {X 0,Y 399.957,Z 1252.781,A -85,B 0,C 180,E1 18454.294,E2 18454.294} C_VEL
LIN {X 0,Y 399.942,Z 1253.493,A -85,B 0,C 180,E1 18452.565,E2 18452.565} C_VEL
LIN {X 0,Y 398.939,Z 1253.73,A -85,B 0,C 180,E1 18451.462,E2 18451.462} C_VEL
LIN {X 0,Y 394.309,Z 1254.018,A -85,B 0,C 180,E1 18449.381,E2 18449.381} C_VEL
LIN {X 0,Y 392.083,Z 1253.853,A -85,B 0,C 180,E1 18447.947,E2 18447.947} C_VEL
LIN {X 0,Y 391.943,Z 1253.792,A -85,B 0,C 180,E1 18447.539,E2 18447.539} C_VEL
LIN {X 0,Y 392.02,Z 1252.116,A -85,B 0,C 180,E1 18443.697,E2 18443.697} C_VEL
LIN {X 0,Y 392.19,Z 1249.344,A -85,B 0,C 180,E1 18440.307,E2 18440.307} C_VEL
LIN {X 0,Y 392.706,Z 1245.593,A -85,B 0,C 180,E1 18437.046,E2 18437.046} C_VEL
LIN {X 0,Y 393.569,Z 1240.97,A -85,B 0,C 180,E1 18433.917,E2 18433.917} C_VEL
LIN {X 0,Y 394.916,Z 1235.286,A -85,B 0,C 180,E1 18430.777,E2 18430.777} C_VEL
LIN {X 0,Y 397,Z 1228.151,A -85,B 0,C 180,E1 18427.485,E2 18427.485} C_VEL
LIN {X 0,Y 400.573,Z 1217.627,A -85,B 0,C 180,E1 18423.455,E2 18423.455} C_VEL
LIN {X 0,Y 404.619,Z 1206.907,A -85,B 0,C 180,E1 18420.049,E2 18420.049} C_VEL
LIN {X 0,Y 408.691,Z 1196.844,A -85,B 0,C 180,E1 18417.264,E2 18417.264} C_VEL
LIN {X 0,Y 413.513,Z 1185.552,A -85,B 0,C 180,E1 18414.521,E2 18414.521} C_VEL
LIN {X 0,Y 420.027,Z 1170.861,A -85,B 0,C 180,E1 18411.408,E2 18411.408} C_VEL
LIN {X 0,Y 427.45,Z 1153.921,A -85,B 0,C 180,E1 18408.364,E2 18408.364} C_VEL
LIN {X 0,Y 434.07,Z 1138.798,A -85,B 0,C 180,E1 18406.007,E2 18406.007} C_VEL
LIN {X 0,Y 440.604,Z 1123.613,A -85,B 0,C 180,E1 18403.923,E2 18403.923} C_VEL
LIN {X 0,Y 447.994,Z 1105.955,A -85,B 0,C 180,E1 18401.796,E2 18401.796} C_VEL
LIN {X 0,Y 457.046,Z 1083,A -85,B 0,C 180,E1 18399.437,E2 18399.437} C_VEL
LIN {X 0,Y 463.899,Z 1064.51,A -85,B 0,C 180,E1 18397.814,E2 18397.814} C_VEL
LIN {X 0,Y 469.998,Z 1046.995,A -85,B 0,C 180,E1 18396.465,E2 18396.465} C_VEL
LIN {X 0,Y 476.016,Z 1028.317,A -85,B 0,C 180,E1 18395.199,E2 18395.199} C_VEL
LIN {X 0,Y 482.558,Z 1006.155,A -85,B 0,C 180,E1 18393.9,E2 18393.9} C_VEL
LIN {X 0,Y 489.258,Z 980.322,A -85,B 0,C 180,E1 18392.644,E2 18392.644} C_VEL
LIN {X 0,Y 494.194,Z 958.237,A -85,B 0,C 180,E1 18391.755,E2 18391.755} C_VEL
LIN {X 0,Y 498.257,Z 937.165,A -85,B 0,C 180,E1 18391.048,E2 18391.048} C_VEL
LIN {X 0,Y 501.758,Z 915.512,A -85,B 0,C 180,E1 18390.454,E2 18390.454} C_VEL
LIN {X 0,Y 505.169,Z 888.921,A -85,B 0,C 180,E1 18389.883,E2 18389.883} C_VEL
LIN {X 0,Y 508.293,Z 846.082,A -85,B 0,C 180,E1 18389.19,E2 18389.19} C_VEL
LIN {X 0,Y 522.809,Z 626.354,A -85,B 0,C 180,E1 18385.774,E2 18385.774} C_VEL
LIN {X 0,Y 525.902,Z 580.791,A -85,B 0,C 180,E1 18385.057,E2 18385.057} C_VEL
LIN {X 0,Y 517.686,Z 568.361,A -85,B 0,C 180,E1 18382.574,E2 18382.574} C_VEL
LIN {X 0,Y 510.335,Z 557.854,A -85,B 0,C 180,E1 18380.052,E2 18380.052} C_VEL
LIN {X 0,Y 504.155,Z 549.2,A -85,B 0,C 180,E1 18377.605,E2 18377.605} C_VEL
LIN {X 0,Y 500.106,Z 543.816,A -85,B 0,C 180,E1 18375.778,E2 18375.778} C_VEL
LIN {X 0,Y 496.513,Z 538.947,A -85,B 0,C 180,E1 18373.925,E2 18373.925} C_VEL
LIN {X 0,Y 493.12,Z 534.245,A -85,B 0,C 180,E1 18371.877,E2 18371.877} C_VEL
LIN {X 0,Y 489.574,Z 530.06,A -85,B 0,C 180,E1 18369.285,E2 18369.285} C_VEL
LIN {X 0,Y 488.599,Z 528.224,A -85,B 0,C 180,E1 18368.355,E2 18368.355} C_VEL
LIN {X 0,Y 485.32,Z 524.618,A -85,B 0,C 180,E1 18364.254,E2 18364.254} C_VEL
LIN {X 0,Y 484.705,Z 522.277,A -85,B 0,C 180,E1 18362.246,E2 18362.246} C_VEL
LIN {X 0,Y 484.779,Z 522.463,A -85,B 0,C 180,E1 18357.872,E2 18357.872} C_VEL
LIN {X 0,Y 486.524,Z 526.586,A -85,B 0,C 180,E1 18354.22,E2 18354.22} C_VEL
LIN {X 0,Y 488.911,Z 528.646,A -85,B 0,C 180,E1 18351.769,E2 18351.769} C_VEL
LIN {X 0,Y 491.392,Z 532.642,A -85,B 0,C 180,E1 18349.685,E2 18349.685} C_VEL
LIN {X 0,Y 493.289,Z 534.56,A -85,B 0,C 180,E1 18348.424,E2 18348.424} C_VEL
LIN {X 0,Y 496.729,Z 539.156,A -85,B 0,C 180,E1 18346.378,E2 18346.378} C_VEL
LIN {X 0,Y 502.131,Z 546.579,A -85,B 0,C 180,E1 18343.694,E2 18343.694} C_VEL
LIN {X 0,Y 509.204,Z 557.431,A -85,B 0,C 180,E1 18340.738,E2 18340.738} C_VEL
LIN {X 0,Y 516.775,Z 569.658,A -85,B 0,C 180,E1 18338.043,E2 18338.043} C_VEL
LIN {X 0,Y 524.165,Z 582.23,A -85,B 0,C 180,E1 18335.727,E2 18335.727} C_VEL
LIN {X 0,Y 525.968,Z 585.57,A -85,B 0,C 180,E1 18335.193,E2 18335.193} C_VEL
LIN {X 0,Y 511.404,Z 804.386,A -85,B 0,C 180,E1 18331.787,E2 18331.787} C_VEL
LIN {X 0,Y 505.206,Z 898.132,A -85,B 0,C 180,E1 18330.309,E2 18330.309} C_VEL
LIN {X 0,Y 502.056,Z 925.986,A -85,B 0,C 180,E1 18329.778,E2 18329.778} C_VEL
LIN {X 0,Y 497.815,Z 951.965,A -85,B 0,C 180,E1 18329.122,E2 18329.122} C_VEL
LIN {X 0,Y 493.693,Z 973.15,A -85,B 0,C 180,E1 18328.452,E2 18328.452} C_VEL
LIN {X 0,Y 489.212,Z 993.188,A -85,B 0,C 180,E1 18327.692,E2 18327.692} C_VEL
LIN {X 0,Y 484.084,Z 1013.57,A -85,B 0,C 180,E1 18326.781,E2 18326.781} C_VEL
LIN {X 0,Y 477.091,Z 1038.605,A -85,B 0,C 180,E1 18325.457,E2 18325.457} C_VEL
LIN {X 0,Y 469.496,Z 1062.453,A -85,B 0,C 180,E1 18323.928,E2 18323.928} C_VEL
LIN {X 0,Y 462.786,Z 1082.069,A -85,B 0,C 180,E1 18322.462,E2 18322.462} C_VEL
LIN {X 0,Y 456.148,Z 1100.338,A -85,B 0,C 180,E1 18320.899,E2 18320.899} C_VEL
LIN {X 0,Y 448.414,Z 1120.581,A -85,B 0,C 180,E1 18318.916,E2 18318.916} C_VEL
LIN {X 0,Y 439.751,Z 1141.954,A -85,B 0,C 180,E1 18316.453,E2 18316.453} C_VEL
LIN {X 0,Y 432.85,Z 1158.541,A -85,B 0,C 180,E1 18314.242,E2 18314.242} C_VEL
LIN {X 0,Y 426.445,Z 1173.766,A -85,B 0,C 180,E1 18311.937,E2 18311.937} C_VEL
LIN {X 0,Y 419.298,Z 1190.889,A -85,B 0,C 180,E1 18308.976,E2 18308.976} C_VEL
LIN {X 0,Y 412.672,Z 1206.801,A -85,B 0,C 180,E1 18305.733,E2 18305.733} C_VEL
LIN {X 0,Y 407.689,Z 1219.221,A -85,B 0,C 180,E1 18302.827,E2 18302.827} C_VEL
LIN {X 0,Y 403.732,Z 1229.749,A -85,B 0,C 180,E1 18300.024,E2 18300.024} C_VEL
LIN {X 0,Y 400,Z 1240.528,A -85,B 0,C 180,E1 18296.746,E2 18296.746} C_VEL
LIN {X 0,Y 396.467,Z 1252.107,A -85,B 0,C 180,E1 18292.547,E2 18292.547} C_VEL
LIN {X 0,Y 394.518,Z 1259.664,A -85,B 0,C 180,E1 18289.243,E2 18289.243} C_VEL
LIN {X 0,Y 393.339,Z 1265.449,A -85,B 0,C 180,E1 18286.244,E2 18286.244} C_VEL
LIN {X 0,Y 392.543,Z 1270.436,A -85,B 0,C 180,E1 18283.109,E2 18283.109} C_VEL
LIN {X 0,Y 392.129,Z 1274.176,A -85,B 0,C 180,E1 18280.14,E2 18280.14} C_VEL
LIN {X 0,Y 391.992,Z 1276.955,A -85,B 0,C 180,E1 18277.186,E2 18277.186} C_VEL
LIN {X 0,Y 391.941,Z 1278.785,A -85,B 0,C 180,E1 18274.249,E2 18274.249} C_VEL
LIN {X 0,Y 391.931,Z 1279.652,A -85,B 0,C 180,E1 18271.468,E2 18271.468} C_VEL
LIN {X 0,Y 391.925,Z 1279.677,A -85,B 0,C 180,E1 18268.691,E2 18268.691} C_VEL
LIN {X 0,Y 391.941,Z 1278.861,A -85,B 0,C 180,E1 18265.911,E2 18265.911} C_VEL
LIN {X 0,Y 391.984,Z 1277.081,A -85,B 0,C 180,E1 18262.974,E2 18262.974} C_VEL
LIN {X 0,Y 392.108,Z 1274.354,A -85,B 0,C 180,E1 18260.022,E2 18260.022} C_VEL
LIN {X 0,Y 392.512,Z 1270.667,A -85,B 0,C 180,E1 18257.053,E2 18257.053} C_VEL
LIN {X 0,Y 393.287,Z 1265.733,A -85,B 0,C 180,E1 18253.919,E2 18253.919} C_VEL
LIN {X 0,Y 394.434,Z 1260,A -85,B 0,C 180,E1 18250.921,E2 18250.921} C_VEL
LIN {X 0,Y 396.351,Z 1252.495,A -85,B 0,C 180,E1 18247.617,E2 18247.617} C_VEL
LIN {X 0,Y 399.55,Z 1241.974,A -85,B 0,C 180,E1 18243.717,E2 18243.717} C_VEL
LIN {X 0,Y 403.53,Z 1230.318,A -85,B 0,C 180,E1 18240.138,E2 18240.138} C_VEL
LIN {X 0,Y 407.452,Z 1219.809,A -85,B 0,C 180,E1 18237.323,E2 18237.323} C_VEL
LIN {X 0,Y 412.106,Z 1208.137,A -85,B 0,C 180,E1 18234.568,E2 18234.568} C_VEL
LIN {X 0,Y 417.808,Z 1194.36,A -85,B 0,C 180,E1 18231.707,E2 18231.707} C_VEL
LIN {X 0,Y 425.695,Z 1175.521,A -85,B 0,C 180,E1 18228.35,E2 18228.35} C_VEL
LIN {X 0,Y 432.411,Z 1159.518,A -85,B 0,C 180,E1 18225.903,E2 18225.903} C_VEL
LIN {X 0,Y 438.95,Z 1143.781,A -85,B 0,C 180,E1 18223.784,E2 18223.784} C_VEL
LIN {X 0,Y 446.484,Z 1125.26,A -85,B 0,C 180,E1 18221.597,E2 18221.597} C_VEL
LIN {X 0,Y 455.339,Z 1102.386,A -85,B 0,C 180,E1 18219.293,E2 18219.293} C_VEL
LIN {X 0,Y 462.469,Z 1082.802,A -85,B 0,C 180,E1 18217.603,E2 18217.603} C_VEL
LIN {X 0,Y 468.79,Z 1064.386,A -85,B 0,C 180,E1 18216.215,E2 18216.215} C_VEL
LIN {X 0,Y 475.308,Z 1044.087,A -85,B 0,C 180,E1 18214.887,E2 18214.887} C_VEL
LIN {X 0,Y 482.548,Z 1019.279,A -85,B 0,C 180,E1 18213.501,E2 18213.501} C_VEL
LIN {X 0,Y 488.642,Z 995.296,A -85,B 0,C 180,E1 18212.4,E2 18212.4} C_VEL
LIN {X 0,Y 493.306,Z 974.641,A -85,B 0,C 180,E1 18211.606,E2 18211.606} C_VEL
LIN {X 0,Y 497.447,Z 953.542,A -85,B 0,C 180,E1 18210.93,E2 18210.93} C_VEL
LIN {X 0,Y 501.156,Z 931.206,A -85,B 0,C 180,E1 18210.35,E2 18210.35} C_VEL
LIN {X 0,Y 504.752,Z 902.604,A -85,B 0,C 180,E1 18209.772,E2 18209.772} C_VEL
LIN {X 0,Y 508.114,Z 854.495,A -85,B 0,C 180,E1 18208.999,E2 18208.999} C_VEL
LIN {X 0,Y 522.319,Z 637.487,A -85,B 0,C 180,E1 18205.62,E2 18205.62} C_VEL
LIN {X 0,Y 525.819,Z 585.189,A -85,B 0,C 180,E1 18204.791,E2 18204.791} C_VEL
LIN {X 0,Y 518.335,Z 572.466,A -85,B 0,C 180,E1 18202.514,E2 18202.514} C_VEL
LIN {X 0,Y 511.002,Z 560.446,A -85,B 0,C 180,E1 18199.995,E2 18199.995} C_VEL
LIN {X 0,Y 504.583,Z 550.598,A -85,B 0,C 180,E1 18197.471,E2 18197.471} C_VEL
LIN {X 0,Y 500.417,Z 544.286,A -85,B 0,C 180,E1 18195.59,E2 18195.59} C_VEL
LIN {X 0,Y 496.229,Z 538.747,A -85,B 0,C 180,E1 18193.458,E2 18193.458} C_VEL
LIN {X 0,Y 492.567,Z 533.81,A -85,B 0,C 180,E1 18191.238,E2 18191.238} C_VEL
LIN {X 0,Y 489.503,Z 530.131,A -85,B 0,C 180,E1 18188.99,E2 18188.99} C_VEL
LIN {X 0,Y 488.444,Z 528.199,A -85,B 0,C 180,E1 18188.002,E2 18188.002} C_VEL
LIN {X 0,Y 485.233,Z 524.729,A -85,B 0,C 180,E1 18184.136,E2 18184.136} C_VEL
LIN {X 0,Y 484.53,Z 522.274,A -85,B 0,C 180,E1 18182.129,E2 18182.129} C_VEL
LIN {X 0,Y 484.633,Z 522.414,A -85,B 0,C 180,E1 18177.043,E2 18177.043} C_VEL
LIN {X 0,Y 485.849,Z 525.782,A -85,B 0,C 180,E1 18174.331,E2 18174.331} C_VEL
LIN {X 0,Y 488.729,Z 528.526,A -85,B 0,C 180,E1 18171.233,E2 18171.233} C_VEL
LIN {X 0,Y 491.315,Z 532.614,A -85,B 0,C 180,E1 18169.09,E2 18169.09} C_VEL
LIN {X 0,Y 493.141,Z 534.473,A -85,B 0,C 180,E1 18167.886,E2 18167.886} C_VEL
LIN {X 0,Y 496.491,Z 539.022,A -85,B 0,C 180,E1 18165.896,E2 18165.896} C_VEL
LIN {X 0,Y 501.554,Z 545.803,A -85,B 0,C 180,E1 18163.377,E2 18163.377} C_VEL
LIN {X 0,Y 505.904,Z 551.84,A -85,B 0,C 180,E1 18161.505,E2 18161.505} C_VEL
LIN {X 0,Y 511.615,Z 559.676,A -85,B 0,C 180,E1 18159.343,E2 18159.343} C_VEL
LIN {X 0,Y 520.654,Z 572.834,A -85,B 0,C 180,E1 18156.366,E2 18156.366} C_VEL
LIN {X 0,Y 525.815,Z 580.993,A -85,B 0,C 180,E1 18154.837,E2 18154.837} C_VEL
LIN {X 0,Y 511.388,Z 796.627,A -85,B 0,C 180,E1 18151.484,E2 18151.484} C_VEL
LIN {X 0,Y 505.681,Z 881.875,A -85,B 0,C 180,E1 18150.141,E2 18150.141} C_VEL
LIN {X 0,Y 502.585,Z 909.549,A -85,B 0,C 180,E1 18149.597,E2 18149.597} C_VEL
LIN {X 0,Y 498.551,Z 935.087,A -85,B 0,C 180,E1 18148.918,E2 18148.918} C_VEL
LIN {X 0,Y 494.517,Z 956.269,A -85,B 0,C 180,E1 18148.221,E2 18148.221} C_VEL
LIN {X 0,Y 489.938,Z 977.071,A -85,B 0,C 180,E1 18147.399,E2 18147.399} C_VEL
LIN {X 0,Y 484.148,Z 1000.124,A -85,B 0,C 180,E1 18146.321,E2 18146.321} C_VEL
LIN {X 0,Y 476.759,Z 1025.776,A -85,B 0,C 180,E1 18144.864,E2 18144.864} C_VEL
LIN {X 0,Y 470.707,Z 1044.692,A -85,B 0,C 180,E1 18143.604,E2 18143.604} C_VEL
LIN {X 0,Y 464.321,Z 1063.142,A -85,B 0,C 180,E1 18142.201,E2 18142.201} C_VEL
LIN {X 0,Y 457.698,Z 1081.092,A -85,B 0,C 180,E1 18140.642,E2 18140.642} C_VEL
LIN {X 0,Y 449.771,Z 1101.507,A -85,B 0,C 180,E1 18138.604,E2 18138.604} C_VEL
LIN {X 0,Y 441.242,Z 1122.027,A -85,B 0,C 180,E1 18136.187,E2 18136.187} C_VEL
LIN {X 0,Y 434.411,Z 1137.925,A -85,B 0,C 180,E1 18134.025,E2 18134.025} C_VEL
LIN {X 0,Y 427.948,Z 1152.702,A -85,B 0,C 180,E1 18131.74,E2 18131.74} C_VEL
LIN {X 0,Y 421.107,Z 1168.315,A -85,B 0,C 180,E1 18128.982,E2 18128.982} C_VEL
LIN {X 0,Y 413.914,Z 1184.633,A -85,B 0,C 180,E1 18125.594,E2 18125.594} C_VEL
LIN {X 0,Y 409.028,Z 1196.015,A -85,B 0,C 180,E1 18122.857,E2 18122.857} C_VEL
LIN {X 0,Y 404.905,Z 1206.162,A -85,B 0,C 180,E1 18120.076,E2 18120.076} C_VEL
LIN {X 0,Y 401.275,Z 1215.615,A -85,B 0,C 180,E1 18117.12,E2 18117.12} C_VEL
LIN {X 0,Y 397.747,Z 1225.866,A -85,B 0,C 180,E1 18113.394,E2 18113.394} C_VEL
LIN {X 0,Y 395.118,Z 1234.544,A -85,B 0,C 180,E1 18109.506,E2 18109.506} C_VEL
LIN {X 0,Y 393.663,Z 1240.56,A -85,B 0,C 180,E1 18106.237,E2 18106.237} C_VEL
LIN {X 0,Y 392.748,Z 1245.287,A -85,B 0,C 180,E1 18103.088,E2 18103.088} C_VEL
LIN {X 0,Y 392.249,Z 1248.797,A -85,B 0,C 180,E1 18100.123,E2 18100.123} C_VEL
LIN {X 0,Y 392.051,Z 1251.397,A -85,B 0,C 180,E1 18097.172,E2 18097.172} C_VEL
LIN {X 0,Y 391.962,Z 1253.11,A -85,B 0,C 180,E1 18094.236,E2 18094.236} C_VEL
LIN {X 0,Y 391.931,Z 1253.949,A -85,B 0,C 180,E1 18091.309,E2 18091.309} C_VEL
LIN {X 0,Y 391.938,Z 1253.917,A -85,B 0,C 180,E1 18088.385,E2 18088.385} C_VEL
LIN {X 0,Y 391.943,Z 1253.792,A -85,B 0,C 180,E1 18087.539,E2 18087.539} C_VEL
LIN {X 0,Y 390.967,Z 1253.555,A -85,B 0,C 180,E1 18086.413,E2 18086.413} C_VEL
LIN {X 0,Y 384.593,Z 1252.131,A -85,B 0,C 180,E1 18083.242,E2 18083.242} C_VEL
LIN {X 0,Y 384.066,Z 1251.539,A -85,B 0,C 180,E1 18082.416,E2 18082.416} C_VEL
LIN {X 0,Y 384.333,Z 1248.836,A -85,B 0,C 180,E1 18079.349,E2 18079.349} C_VEL
LIN {X 0,Y 384.932,Z 1245.059,A -85,B 0,C 180,E1 18076.168,E2 18076.168} C_VEL
LIN {X 0,Y 386.123,Z 1239.514,A -85,B 0,C 180,E1 18072.513,E2 18072.513} C_VEL
LIN {X 0,Y 388.457,Z 1231.171,A -85,B 0,C 180,E1 18068.238,E2 18068.238} C_VEL
LIN {X 0,Y 391,Z 1223.575,A -85,B 0,C 180,E1 18065.037,E2 18065.037} C_VEL
LIN {X 0,Y 394.196,Z 1215.112,A -85,B 0,C 180,E1 18061.972,E2 18061.972} C_VEL
LIN {X 0,Y 398.247,Z 1205.167,A -85,B 0,C 180,E1 18058.849,E2 18058.849} C_VEL
LIN {X 0,Y 404.187,Z 1191.694,A -85,B 0,C 180,E1 18055.217,E2 18055.217} C_VEL
LIN {X 0,Y 410.61,Z 1177.323,A -85,B 0,C 180,E1 18051.964,E2 18051.964} C_VEL
LIN {X 0,Y 416.556,Z 1164.401,A -85,B 0,C 180,E1 18049.415,E2 18049.415} C_VEL
LIN {X 0,Y 422.769,Z 1150.864,A -85,B 0,C 180,E1 18047.061,E2 18047.061} C_VEL
LIN {X 0,Y 430.427,Z 1134.05,A -85,B 0,C 180,E1 18044.502,E2 18044.502} C_VEL
LIN {X 0,Y 439.266,Z 1113.894,A -85,B 0,C 180,E1 18041.892,E2 18041.892} C_VEL
LIN {X 0,Y 446.381,Z 1096.9,A -85,B 0,C 180,E1 18039.992,E2 18039.992} C_VEL
LIN {X 0,Y 453.403,Z 1079.302,A -85,B 0,C 180,E1 18038.266,E2 18038.266} C_VEL
LIN {X 0,Y 460.426,Z 1060.674,A -85,B 0,C 180,E1 18036.67,E2 18036.67} C_VEL
LIN {X 0,Y 468.816,Z 1036.616,A -85,B 0,C 180,E1 18034.904,E2 18034.904} C_VEL
LIN {X 0,Y 475.671,Z 1014.594,A -85,B 0,C 180,E1 18033.549,E2 18033.549} C_VEL
LIN {X 0,Y 481.317,Z 994.579,A -85,B 0,C 180,E1 18032.492,E2 18032.492} C_VEL
LIN {X 0,Y 486.469,Z 974.193,A -85,B 0,C 180,E1 18031.569,E2 18031.569} C_VEL
LIN {X 0,Y 491.451,Z 951.66,A -85,B 0,C 180,E1 18030.709,E2 18030.709} C_VEL
LIN {X 0,Y 496.652,Z 922.902,A -85,B 0,C 180,E1 18029.837,E2 18029.837} C_VEL
LIN {X 0,Y 499.856,Z 900.239,A -85,B 0,C 180,E1 18029.31,E2 18029.31} C_VEL
LIN {X 0,Y 502.187,Z 878.025,A -85,B 0,C 180,E1 18028.901,E2 18028.901} C_VEL
LIN {X 0,Y 516.841,Z 662.858,A -85,B 0,C 180,E1 18025.541,E2 18025.541} C_VEL
LIN {X 0,Y 522.247,Z 585.782,A -85,B 0,C 180,E1 18024.341,E2 18024.341} C_VEL
LIN {X 0,Y 515.148,Z 574.951,A -85,B 0,C 180,E1 18022.12,E2 18022.12} C_VEL
LIN {X 0,Y 508.185,Z 564.818,A -85,B 0,C 180,E1 18019.661,E2 18019.661} C_VEL
LIN {X 0,Y 502.271,Z 556.44,A -85,B 0,C 180,E1 18017.255,E2 18017.255} C_VEL
LIN {X 0,Y 498.432,Z 551.236,A -85,B 0,C 180,E1 18015.474,E2 18015.474} C_VEL
LIN {X 0,Y 495.02,Z 546.54,A -85,B 0,C 180,E1 18013.67,E2 18013.67} C_VEL
LIN {X 0,Y 491.353,Z 541.532,A -85,B 0,C 180,E1 18011.385,E2 18011.385} C_VEL
LIN {X 0,Y 488.206,Z 537.51,A -85,B 0,C 180,E1 18008.955,E2 18008.955} C_VEL
LIN {X 0,Y 487.369,Z 536.039,A -85,B 0,C 180,E1 18008.138,E2 18008.138} C_VEL
LIN {X 0,Y 484.235,Z 532.362,A -85,B 0,C 180,E1 18004.026,E2 18004.026} C_VEL
LIN {X 0,Y 483.697,Z 530.211,A -85,B 0,C 180,E1 18002.132,E2 18002.132} C_VEL
LIN {X 0,Y 483.792,Z 530.503,A -85,B 0,C 180,E1 17997.868,E2 17997.868} C_VEL
LIN {X 0,Y 485.549,Z 534.568,A -85,B 0,C 180,E1 17994.209,E2 17994.209} C_VEL
LIN {X 0,Y 487.742,Z 536.47,A -85,B 0,C 180,E1 17991.927,E2 17991.927} C_VEL
LIN {X 0,Y 490.257,Z 540.528,A -85,B 0,C 180,E1 17989.779,E2 17989.779} C_VEL
LIN {X 0,Y 492.04,Z 542.41,A -85,B 0,C 180,E1 17988.572,E2 17988.572} C_VEL
LIN {X 0,Y 496.146,Z 548.085,A -85,B 0,C 180,E1 17986.124,E2 17986.124} C_VEL
LIN {X 0,Y 500.655,Z 554.299,A -85,B 0,C 180,E1 17983.883,E2 17983.883} C_VEL
LIN {X 0,Y 507.424,Z 564.929,A -85,B 0,C 180,E1 17980.996,E2 17980.996} C_VEL
LIN {X 0,Y 514.571,Z 576.673,A -85,B 0,C 180,E1 17978.394,E2 17978.394} C_VEL
LIN {X 0,Y 521.671,Z 588.97,A -85,B 0,C 180,E1 17976.112,E2 17976.112} C_VEL
LIN {X 0,Y 522.281,Z 590.368,A -85,B 0,C 180,E1 17975.917,E2 17975.917} C_VEL
LIN {X 0,Y 507.212,Z 810.695,A -85,B 0,C 180,E1 17972.486,E2 17972.486} C_VEL
LIN {X 0,Y 501.248,Z 898.102,A -85,B 0,C 180,E1 17971.105,E2 17971.105} C_VEL
LIN {X 0,Y 497.985,Z 926.126,A -85,B 0,C 180,E1 17970.57,E2 17970.57} C_VEL
LIN {X 0,Y 493.718,Z 951.709,A -85,B 0,C 180,E1 17969.926,E2 17969.926} C_VEL
LIN {X 0,Y 489.498,Z 972.892,A -85,B 0,C 180,E1 17969.261,E2 17969.261} C_VEL
LIN {X 0,Y 484.913,Z 992.928,A -85,B 0,C 180,E1 17968.504,E2 17968.504} C_VEL
LIN {X 0,Y 479.657,Z 1013.309,A -85,B 0,C 180,E1 17967.598,E2 17967.598} C_VEL
LIN {X 0,Y 472.482,Z 1038.341,A -85,B 0,C 180,E1 17966.277,E2 17966.277} C_VEL
LIN {X 0,Y 464.686,Z 1062.187,A -85,B 0,C 180,E1 17964.75,E2 17964.75} C_VEL
LIN {X 0,Y 457.799,Z 1081.775,A -85,B 0,C 180,E1 17963.286,E2 17963.286} C_VEL
LIN {X 0,Y 450.95,Z 1100.069,A -85,B 0,C 180,E1 17961.719,E2 17961.719} C_VEL
LIN {X 0,Y 443.368,Z 1119.291,A -85,B 0,C 180,E1 17959.835,E2 17959.835} C_VEL
LIN {X 0,Y 434.133,Z 1141.418,A -85,B 0,C 180,E1 17957.289,E2 17957.289} C_VEL
LIN {X 0,Y 427.059,Z 1157.828,A -85,B 0,C 180,E1 17955.092,E2 17955.092} C_VEL
LIN {X 0,Y 420.588,Z 1172.633,A -85,B 0,C 180,E1 17952.843,E2 17952.843} C_VEL
LIN {X 0,Y 414.003,Z 1187.653,A -85,B 0,C 180,E1 17950.253,E2 17950.253} C_VEL
LIN {X 0,Y 406.391,Z 1205.23,A -85,B 0,C 180,E1 17946.724,E2 17946.724} C_VEL
LIN {X 0,Y 400.874,Z 1218.36,A -85,B 0,C 180,E1 17943.629,E2 17943.629} C_VEL
LIN {X 0,Y 396.543,Z 1229.238,A -85,B 0,C 180,E1 17940.701,E2 17940.701} C_VEL
LIN {X 0,Y 392.833,Z 1239.314,A -85,B 0,C 180,E1 17937.603,E2 17937.603} C_VEL
LIN {X 0,Y 389.217,Z 1250.381,A -85,B 0,C 180,E1 17933.632,E2 17933.632} C_VEL
LIN {X 0,Y 386.779,Z 1259.125,A -85,B 0,C 180,E1 17929.779,E2 17929.779} C_VEL
LIN {X 0,Y 385.44,Z 1265.18,A -85,B 0,C 180,E1 17926.586,E2 17926.586} C_VEL
LIN {X 0,Y 384.596,Z 1270.168,A -85,B 0,C 180,E1 17923.385,E2 17923.385} C_VEL
LIN {X 0,Y 384.149,Z 1273.969,A -85,B 0,C 180,E1 17920.299,E2 17920.299} C_VEL
LIN {X 0,Y 383.993,Z 1276.808,A -85,B 0,C 180,E1 17917.187,E2 17917.187} C_VEL
LIN {X 0,Y 383.945,Z 1278.631,A -85,B 0,C 180,E1 17914.106,E2 17914.106} C_VEL
LIN {X 0,Y 383.915,Z 1279.459,A -85,B 0,C 180,E1 17911.051,E2 17911.051} C_VEL
LIN {X 0,Y 383.943,Z 1279.321,A -85,B 0,C 180,E1 17908.067,E2 17908.067} C_VEL
LIN {X 0,Y 383.949,Z 1278.173,A -85,B 0,C 180,E1 17904.927,E2 17904.927} C_VEL
LIN {X 0,Y 384.047,Z 1275.636,A -85,B 0,C 180,E1 17901.322,E2 17901.322} C_VEL
LIN {X 0,Y 384.458,Z 1271.251,A -85,B 0,C 180,E1 17897.389,E2 17897.389} C_VEL
LIN {X 0,Y 385.291,Z 1265.987,A -85,B 0,C 180,E1 17893.886,E2 17893.886} C_VEL
LIN {X 0,Y 386.546,Z 1260.039,A -85,B 0,C 180,E1 17890.673,E2 17890.673} C_VEL
LIN {X 0,Y 388.44,Z 1252.947,A -85,B 0,C 180,E1 17887.455,E2 17887.455} C_VEL
LIN {X 0,Y 391.291,Z 1243.829,A -85,B 0,C 180,E1 17883.936,E2 17883.936} C_VEL
LIN {X 0,Y 395.85,Z 1231.092,A -85,B 0,C 180,E1 17879.833,E2 17879.833} C_VEL
LIN {X 0,Y 400.36,Z 1219.57,A -85,B 0,C 180,E1 17876.681,E2 17876.681} C_VEL
LIN {X 0,Y 405.249,Z 1207.858,A -85,B 0,C 180,E1 17873.875,E2 17873.875} C_VEL
LIN {X 0,Y 411.196,Z 1194.08,A -85,B 0,C 180,E1 17870.976,E2 17870.976} C_VEL
LIN {X 0,Y 419.423,Z 1175.242,A -85,B 0,C 180,E1 17867.584,E2 17867.584} C_VEL
LIN {X 0,Y 426.405,Z 1159.239,A -85,B 0,C 180,E1 17865.116,E2 17865.116} C_VEL
LIN {X 0,Y 433.183,Z 1143.503,A -85,B 0,C 180,E1 17862.982,E2 17862.982} C_VEL
LIN {X 0,Y 440.977,Z 1124.983,A -85,B 0,C 180,E1 17860.784,E2 17860.784} C_VEL
LIN {X 0,Y 450.203,Z 1101.884,A -85,B 0,C 180,E1 17858.453,E2 17858.453} C_VEL
LIN {X 0,Y 457.386,Z 1082.731,A -85,B 0,C 180,E1 17856.798,E2 17856.798} C_VEL
LIN {X 0,Y 463.967,Z 1064.083,A -85,B 0,C 180,E1 17855.39,E2 17855.39} C_VEL
LIN {X 0,Y 470.648,Z 1043.812,A -85,B 0,C 180,E1 17854.064,E2 17854.064} C_VEL
LIN {X 0,Y 478.083,Z 1019.003,A -85,B 0,C 180,E1 17852.684,E2 17852.684} C_VEL
LIN {X 0,Y 484.352,Z 994.925,A -85,B 0,C 180,E1 17851.583,E2 17851.583} C_VEL
LIN {X 0,Y 489.102,Z 974.366,A -85,B 0,C 180,E1 17850.797,E2 17850.797} C_VEL
LIN {X 0,Y 493.366,Z 953.134,A -85,B 0,C 180,E1 17850.12,E2 17850.12} C_VEL
LIN {X 0,Y 497.154,Z 930.799,A -85,B 0,C 180,E1 17849.545,E2 17849.545} C_VEL
LIN {X 0,Y 500.838,Z 901.89,A -85,B 0,C 180,E1 17848.965,E2 17848.965} C_VEL
LIN {X 0,Y 504.37,Z 852.495,A -85,B 0,C 180,E1 17848.172,E2 17848.172} C_VEL
LIN {X 0,Y 518.997,Z 635.545,A -85,B 0,C 180,E1 17844.791,E2 17844.791} C_VEL
LIN {X 0,Y 522.15,Z 589.992,A -85,B 0,C 180,E1 17844.072,E2 17844.072} C_VEL
LIN {X 0,Y 515.697,Z 578.822,A -85,B 0,C 180,E1 17842.035,E2 17842.035} C_VEL
LIN {X 0,Y 508.831,Z 567.372,A -85,B 0,C 180,E1 17839.605,E2 17839.605} C_VEL
LIN {X 0,Y 502.687,Z 557.767,A -85,B 0,C 180,E1 17837.121,E2 17837.121} C_VEL
LIN {X 0,Y 498.845,Z 551.846,A -85,B 0,C 180,E1 17835.342,E2 17835.342} C_VEL
LIN {X 0,Y 494.84,Z 546.44,A -85,B 0,C 180,E1 17833.258,E2 17833.258} C_VEL
LIN {X 0,Y 491.24,Z 541.546,A -85,B 0,C 180,E1 17831.031,E2 17831.031} C_VEL
LIN {X 0,Y 488.253,Z 537.818,A -85,B 0,C 180,E1 17828.776,E2 17828.776} C_VEL
LIN {X 0,Y 487.342,Z 536.088,A -85,B 0,C 180,E1 17827.901,E2 17827.901} C_VEL
LIN {X 0,Y 484.192,Z 532.608,A -85,B 0,C 180,E1 17824.026,E2 17824.026} C_VEL
LIN {X 0,Y 483.516,Z 530.209,A -85,B 0,C 180,E1 17822.015,E2 17822.015} C_VEL
LIN {X 0,Y 483.62,Z 530.3,A -85,B 0,C 180,E1 17817.156,E2 17817.156} C_VEL
LIN {X 0,Y 484.793,Z 533.662,A -85,B 0,C 180,E1 17814.437,E2 17814.437} C_VEL
LIN {X 0,Y 487.615,Z 536.492,A -85,B 0,C 180,E1 17811.331,E2 17811.331} C_VEL
LIN {X 0,Y 490.18,Z 540.5,A -85,B 0,C 180,E1 17809.183,E2 17809.183} C_VEL
LIN {X 0,Y 491.891,Z 542.33,A -85,B 0,C 180,E1 17808.033,E2 17808.033} C_VEL
LIN {X 0,Y 495.311,Z 546.924,A -85,B 0,C 180,E1 17805.981,E2 17805.981} C_VEL
LIN {X 0,Y 500.201,Z 553.716,A -85,B 0,C 180,E1 17803.51,E2 17803.51} C_VEL
LIN {X 0,Y 504.114,Z 559.204,A -85,B 0,C 180,E1 17801.796,E2 17801.796} C_VEL
LIN {X 0,Y 509.728,Z 567.054,A -85,B 0,C 180,E1 17799.623,E2 17799.623} C_VEL
LIN {X 0,Y 518.468,Z 579.989,A -85,B 0,C 180,E1 17796.682,E2 17796.682} C_VEL
LIN {X 0,Y 522.127,Z 585.953,A -85,B 0,C 180,E1 17795.559,E2 17795.559} C_VEL
LIN {X 0,Y 507.351,Z 800.89,A -85,B 0,C 180,E1 17792.216,E2 17792.216} C_VEL
LIN {X 0,Y 501.726,Z 882.374,A -85,B 0,C 180,E1 17790.93,E2 17790.93} C_VEL
LIN {X 0,Y 498.495,Z 910.346,A -85,B 0,C 180,E1 17790.379,E2 17790.379} C_VEL
LIN {X 0,Y 494.454,Z 935.362,A -85,B 0,C 180,E1 17789.715,E2 17789.715} C_VEL
LIN {X 0,Y 490.326,Z 956.543,A -85,B 0,C 180,E1 17789.021,E2 17789.021} C_VEL
LIN {X 0,Y 485.723,Z 976.985,A -85,B 0,C 180,E1 17788.216,E2 17788.216} C_VEL
LIN {X 0,Y 480.027,Z 999.163,A -85,B 0,C 180,E1 17787.187,E2 17787.187} C_VEL
LIN {X 0,Y 472.512,Z 1024.874,A -85,B 0,C 180,E1 17785.744,E2 17785.744} C_VEL
LIN {X 0,Y 465.91,Z 1044.966,A -85,B 0,C 180,E1 17784.412,E2 17784.412} C_VEL
LIN {X 0,Y 459.345,Z 1063.416,A -85,B 0,C 180,E1 17783.009,E2 17783.009} C_VEL
LIN {X 0,Y 452.535,Z 1081.366,A -85,B 0,C 180,E1 17781.446,E2 17781.446} C_VEL
LIN {X 0,Y 444.384,Z 1101.722,A -85,B 0,C 180,E1 17779.408,E2 17779.408} C_VEL
LIN {X 0,Y 435.546,Z 1122.302,A -85,B 0,C 180,E1 17776.973,E2 17776.973} C_VEL
LIN {X 0,Y 428.473,Z 1138.201,A -85,B 0,C 180,E1 17774.797,E2 17774.797} C_VEL
LIN {X 0,Y 421.771,Z 1152.978,A -85,B 0,C 180,E1 17772.493,E2 17772.493} C_VEL
LIN {X 0,Y 414.326,Z 1169.349,A -85,B 0,C 180,E1 17769.566,E2 17769.566} C_VEL
LIN {X 0,Y 407.163,Z 1184.909,A -85,B 0,C 180,E1 17766.277,E2 17766.277} C_VEL
LIN {X 0,Y 401.798,Z 1196.852,A -85,B 0,C 180,E1 17763.355,E2 17763.355} C_VEL
LIN {X 0,Y 397.5,Z 1206.941,A -85,B 0,C 180,E1 17760.529,E2 17760.529} C_VEL
LIN {X 0,Y 393.552,Z 1216.785,A -85,B 0,C 180,E1 17757.369,E2 17757.369} C_VEL
LIN {X 0,Y 389.661,Z 1227.559,A -85,B 0,C 180,E1 17753.268,E2 17753.268} C_VEL
LIN {X 0,Y 387.28,Z 1235.11,A -85,B 0,C 180,E1 17749.76,E2 17749.76} C_VEL
LIN {X 0,Y 385.801,Z 1240.865,A -85,B 0,C 180,E1 17746.556,E2 17746.556} C_VEL
LIN {X 0,Y 384.828,Z 1245.555,A -85,B 0,C 180,E1 17743.363,E2 17743.363} C_VEL
LIN {X 0,Y 384.294,Z 1249.063,A -85,B 0,C 180,E1 17740.335,E2 17740.335} C_VEL
LIN {X 0,Y 384.063,Z 1251.686,A -85,B 0,C 180,E1 17737.288,E2 17737.288} C_VEL
LIN {X 0,Y 383.968,Z 1253.374,A -85,B 0,C 180,E1 17734.324,E2 17734.324} C_VEL
LIN {X 0,Y 383.943,Z 1254.189,A -85,B 0,C 180,E1 17731.485,E2 17731.485} C_VEL
LIN {X 0,Y 383.93,Z 1254.223,A -85,B 0,C 180,E1 17728.65,E2 17728.65} C_VEL
LIN {X 0,Y 383.969,Z 1253.409,A -85,B 0,C 180,E1 17725.662,E2 17725.662} C_VEL
LIN {X 0,Y 384.063,Z 1251.72,A -85,B 0,C 180,E1 17722.664,E2 17722.664} C_VEL
LIN {X 0,Y 384.066,Z 1251.539,A -85,B 0,C 180,E1 17722.416,E2 17722.416} C_VEL
LIN {X 0,Y 383.114,Z 1250.768,A -85,B 0,C 180,E1 17721.271,E2 17721.271} C_VEL
LIN {X 0,Y 377.091,Z 1248.035,A -85,B 0,C 180,E1 17718.042,E2 17718.042} C_VEL
LIN {X 0,Y 376.708,Z 1247.051,A -85,B 0,C 180,E1 17717.209,E2 17717.209} C_VEL
LIN {X 0,Y 377.748,Z 1241.998,A -85,B 0,C 180,E1 17713.541,E2 17713.541} C_VEL
LIN {X 0,Y 379.234,Z 1236.406,A -85,B 0,C 180,E1 17710.267,E2 17710.267} C_VEL
LIN {X 0,Y 381.436,Z 1229.594,A -85,B 0,C 180,E1 17706.942,E2 17706.942} C_VEL
LIN {X 0,Y 384.595,Z 1221.067,A -85,B 0,C 180,E1 17703.425,E2 17703.425} C_VEL
LIN {X 0,Y 389.612,Z 1208.961,A -85,B 0,C 180,E1 17699.283,E2 17699.283} C_VEL
LIN {X 0,Y 394.494,Z 1197.949,A -85,B 0,C 180,E1 17696.103,E2 17696.103} C_VEL
LIN {X 0,Y 399.748,Z 1186.718,A -85,B 0,C 180,E1 17693.281,E2 17693.281} C_VEL
LIN {X 0,Y 405.912,Z 1173.821,A -85,B 0,C 180,E1 17690.446,E2 17690.446} C_VEL
LIN {X 0,Y 414.38,Z 1156.125,A -85,B 0,C 180,E1 17687.115,E2 17687.115} C_VEL
LIN {X 0,Y 421.932,Z 1140.049,A -85,B 0,C 180,E1 17684.544,E2 17684.544} C_VEL
LIN {X 0,Y 429.097,Z 1124.515,A -85,B 0,C 180,E1 17682.376,E2 17682.376} C_VEL
LIN {X 0,Y 436.663,Z 1107.586,A -85,B 0,C 180,E1 17680.308,E2 17680.308} C_VEL
LIN {X 0,Y 446.26,Z 1084.851,A -85,B 0,C 180,E1 17677.932,E2 17677.932} C_VEL
LIN {X 0,Y 453.759,Z 1065.765,A -85,B 0,C 180,E1 17676.239,E2 17676.239} C_VEL
LIN {X 0,Y 460.512,Z 1047.42,A -85,B 0,C 180,E1 17674.823,E2 17674.823} C_VEL
LIN {X 0,Y 466.537,Z 1029.732,A -85,B 0,C 180,E1 17673.624,E2 17673.624} C_VEL
LIN {X 0,Y 472.762,Z 1009.766,A -85,B 0,C 180,E1 17672.443,E2 17672.443} C_VEL
LIN {X 0,Y 479.82,Z 984.664,A -85,B 0,C 180,E1 17671.187,E2 17671.187} C_VEL
LIN {X 0,Y 485.756,Z 959.457,A -85,B 0,C 180,E1 17670.165,E2 17670.165} C_VEL
LIN {X 0,Y 490.05,Z 938.272,A -85,B 0,C 180,E1 17669.457,E2 17669.457} C_VEL
LIN {X 0,Y 493.658,Z 917.049,A -85,B 0,C 180,E1 17668.875,E2 17668.875} C_VEL
LIN {X 0,Y 496.848,Z 893.602,A -85,B 0,C 180,E1 17668.365,E2 17668.365} C_VEL
LIN {X 0,Y 499.916,Z 857.814,A -85,B 0,C 180,E1 17667.765,E2 17667.765} C_VEL
LIN {X 0,Y 515.315,Z 636.948,A -85,B 0,C 180,E1 17664.329,E2 17664.329} C_VEL
LIN {X 0,Y 518.593,Z 590.614,A -85,B 0,C 180,E1 17663.589,E2 17663.589} C_VEL
LIN {X 0,Y 510.429,Z 578.109,A -85,B 0,C 180,E1 17660.887,E2 17660.887} C_VEL
LIN {X 0,Y 504.01,Z 568.79,A -85,B 0,C 180,E1 17658.447,E2 17658.447} C_VEL
LIN {X 0,Y 499.547,Z 562.529,A -85,B 0,C 180,E1 17656.513,E2 17656.513} C_VEL
LIN {X 0,Y 496.884,Z 558.789,A -85,B 0,C 180,E1 17655.225,E2 17655.225} C_VEL
LIN {X 0,Y 493.538,Z 554.128,A -85,B 0,C 180,E1 17653.413,E2 17653.413} C_VEL
LIN {X 0,Y 490.038,Z 549.265,A -85,B 0,C 180,E1 17651.177,E2 17651.177} C_VEL
LIN {X 0,Y 486.972,Z 545.2,A -85,B 0,C 180,E1 17648.74,E2 17648.74} C_VEL
LIN {X 0,Y 486.273,Z 543.927,A -85,B 0,C 180,E1 17648.038,E2 17648.038} C_VEL
LIN {X 0,Y 483.204,Z 540.241,A -85,B 0,C 180,E1 17643.916,E2 17643.916} C_VEL
LIN {X 0,Y 482.691,Z 538.146,A -85,B 0,C 180,E1 17642.018,E2 17642.018} C_VEL
LIN {X 0,Y 482.785,Z 538.384,A -85,B 0,C 180,E1 17637.982,E2 17637.982} C_VEL
LIN {X 0,Y 484.483,Z 542.448,A -85,B 0,C 180,E1 17634.315,E2 17634.315} C_VEL
LIN {X 0,Y 486.631,Z 544.426,A -85,B 0,C 180,E1 17632.028,E2 17632.028} C_VEL
LIN {X 0,Y 489.284,Z 548.581,A -85,B 0,C 180,E1 17629.759,E2 17629.759} C_VEL
LIN {X 0,Y 490.795,Z 550.256,A -85,B 0,C 180,E1 17628.721,E2 17628.721} C_VEL
LIN {X 0,Y 494.743,Z 555.796,A -85,B 0,C 180,E1 17626.322,E2 17626.322} C_VEL
LIN {X 0,Y 499.185,Z 562.017,A -85,B 0,C 180,E1 17624.073,E2 17624.073} C_VEL
LIN {X 0,Y 505.857,Z 572.775,A -85,B 0,C 180,E1 17621.175,E2 17621.175} C_VEL
LIN {X 0,Y 512.613,Z 584.103,A -85,B 0,C 180,E1 17618.667,E2 17618.667} C_VEL
LIN {X 0,Y 518.701,Z 594.779,A -85,B 0,C 180,E1 17616.658,E2 17616.658} C_VEL
LIN {X 0,Y 503.455,Z 811.73,A -85,B 0,C 180,E1 17613.279,E2 17613.279} C_VEL
LIN {X 0,Y 497.407,Z 897.857,A -85,B 0,C 180,E1 17611.917,E2 17611.917} C_VEL
LIN {X 0,Y 494.056,Z 926.004,A -85,B 0,C 180,E1 17611.38,E2 17611.38} C_VEL
LIN {X 0,Y 489.721,Z 951.454,A -85,B 0,C 180,E1 17610.744,E2 17610.744} C_VEL
LIN {X 0,Y 485.404,Z 972.635,A -85,B 0,C 180,E1 17610.083,E2 17610.083} C_VEL
LIN {X 0,Y 480.714,Z 992.669,A -85,B 0,C 180,E1 17609.331,E2 17609.331} C_VEL
LIN {X 0,Y 475.175,Z 1013.617,A -85,B 0,C 180,E1 17608.402,E2 17608.402} C_VEL
LIN {X 0,Y 467.67,Z 1038.997,A -85,B 0,C 180,E1 17607.058,E2 17607.058} C_VEL
LIN {X 0,Y 459.942,Z 1062.018,A -85,B 0,C 180,E1 17605.582,E2 17605.582} C_VEL
LIN {X 0,Y 453.18,Z 1080.766,A -85,B 0,C 180,E1 17604.184,E2 17604.184} C_VEL
LIN {X 0,Y 446.375,Z 1098.451,A -85,B 0,C 180,E1 17602.68,E2 17602.68} C_VEL
LIN {X 0,Y 439.103,Z 1116.348,A -85,B 0,C 180,E1 17600.946,E2 17600.946} C_VEL
LIN {X 0,Y 430.17,Z 1137.457,A -85,B 0,C 180,E1 17598.581,E2 17598.581} C_VEL
LIN {X 0,Y 421.608,Z 1156.585,A -85,B 0,C 180,E1 17596.042,E2 17596.042} C_VEL
LIN {X 0,Y 414.838,Z 1171.5,A -85,B 0,C 180,E1 17593.775,E2 17593.775} C_VEL
LIN {X 0,Y 408.47,Z 1185.429,A -85,B 0,C 180,E1 17591.376,E2 17591.376} C_VEL
LIN {X 0,Y 402.105,Z 1199.478,A -85,B 0,C 180,E1 17588.625,E2 17588.625} C_VEL
LIN {X 0,Y 394.645,Z 1216.328,A -85,B 0,C 180,E1 17584.761,E2 17584.761} C_VEL
LIN {X 0,Y 389.655,Z 1228.146,A -85,B 0,C 180,E1 17581.572,E2 17581.572} C_VEL
LIN {X 0,Y 385.733,Z 1238.099,A -85,B 0,C 180,E1 17578.493,E2 17578.493} C_VEL
LIN {X 0,Y 382.472,Z 1247.267,A -85,B 0,C 180,E1 17575.228,E2 17575.228} C_VEL
LIN {X 0,Y 379.484,Z 1257.001,A -85,B 0,C 180,E1 17571.133,E2 17571.133} C_VEL
LIN {X 0,Y 377.658,Z 1264.385,A -85,B 0,C 180,E1 17567.256,E2 17567.256} C_VEL
LIN {X 0,Y 376.718,Z 1269.473,A -85,B 0,C 180,E1 17563.983,E2 17563.983} C_VEL
LIN {X 0,Y 376.227,Z 1273.314,A -85,B 0,C 180,E1 17560.883,E2 17560.883} C_VEL
LIN {X 0,Y 375.991,Z 1276.19,A -85,B 0,C 180,E1 17557.801,E2 17557.801} C_VEL
LIN {X 0,Y 375.95,Z 1278.047,A -85,B 0,C 180,E1 17554.889,E2 17554.889} C_VEL
LIN {X 0,Y 375.946,Z 1279.08,A -85,B 0,C 180,E1 17551.836,E2 17551.836} C_VEL
LIN {X 0,Y 375.92,Z 1279.198,A -85,B 0,C 180,E1 17548.94,E2 17548.94} C_VEL
LIN {X 0,Y 375.948,Z 1278.385,A -85,B 0,C 180,E1 17545.847,E2 17545.847} C_VEL
LIN {X 0,Y 375.993,Z 1276.586,A -85,B 0,C 180,E1 17542.718,E2 17542.718} C_VEL
LIN {X 0,Y 376.165,Z 1273.806,A -85,B 0,C 180,E1 17539.58,E2 17539.58} C_VEL
LIN {X 0,Y 376.617,Z 1270.13,A -85,B 0,C 180,E1 17536.497,E2 17536.497} C_VEL
LIN {X 0,Y 377.491,Z 1265.192,A -85,B 0,C 180,E1 17533.227,E2 17533.227} C_VEL
LIN {X 0,Y 378.902,Z 1259.142,A -85,B 0,C 180,E1 17529.945,E2 17529.945} C_VEL
LIN {X 0,Y 381.203,Z 1251.219,A -85,B 0,C 180,E1 17526.348,E2 17526.348} C_VEL
LIN {X 0,Y 385.052,Z 1240.011,A -85,B 0,C 180,E1 17522.143,E2 17522.143} C_VEL
LIN {X 0,Y 389.06,Z 1229.587,A -85,B 0,C 180,E1 17518.85,E2 17518.85} C_VEL
LIN {X 0,Y 393.596,Z 1218.706,A -85,B 0,C 180,E1 17515.856,E2 17515.856} C_VEL
LIN {X 0,Y 399.017,Z 1206.282,A -85,B 0,C 180,E1 17512.86,E2 17512.86} C_VEL
LIN {X 0,Y 406.347,Z 1190.148,A -85,B 0,C 180,E1 17509.495,E2 17509.495} C_VEL
LIN {X 0,Y 414.01,Z 1173.245,A -85,B 0,C 180,E1 17506.515,E2 17506.515} C_VEL
LIN {X 0,Y 420.717,Z 1158.453,A -85,B 0,C 180,E1 17504.234,E2 17504.234} C_VEL
LIN {X 0,Y 427.741,Z 1142.711,A -85,B 0,C 180,E1 17502.095,E2 17502.095} C_VEL
LIN {X 0,Y 436.064,Z 1123.581,A -85,B 0,C 180,E1 17499.825,E2 17499.825} C_VEL
LIN {X 0,Y 445.254,Z 1101.157,A -85,B 0,C 180,E1 17497.574,E2 17497.574} C_VEL
LIN {X 0,Y 452.514,Z 1082.353,A -85,B 0,C 180,E1 17495.95,E2 17495.95} C_VEL
LIN {X 0,Y 459.325,Z 1063.558,A -85,B 0,C 180,E1 17494.533,E2 17494.533} C_VEL
LIN {X 0,Y 466.417,Z 1042.539,A -85,B 0,C 180,E1 17493.165,E2 17493.165} C_VEL
LIN {X 0,Y 474.328,Z 1016.453,A -85,B 0,C 180,E1 17491.741,E2 17491.741} C_VEL
LIN {X 0,Y 480.316,Z 993.94,A -85,B 0,C 180,E1 17490.727,E2 17490.727} C_VEL
LIN {X 0,Y 485.16,Z 973.347,A -85,B 0,C 180,E1 17489.948,E2 17489.948} C_VEL
LIN {X 0,Y 489.619,Z 951.523,A -85,B 0,C 180,E1 17489.264,E2 17489.264} C_VEL
LIN {X 0,Y 493.931,Z 926.207,A -85,B 0,C 180,E1 17488.63,E2 17488.63} C_VEL
LIN {X 0,Y 497.303,Z 897.953,A -85,B 0,C 180,E1 17488.09,E2 17488.09} C_VEL
LIN {X 0,Y 503.357,Z 811.666,A -85,B 0,C 180,E1 17486.726,E2 17486.726} C_VEL
LIN {X 0,Y 518.58,Z 594.891,A -85,B 0,C 180,E1 17483.351,E2 17483.351} C_VEL
LIN {X 0,Y 513.33,Z 585.568,A -85,B 0,C 180,E1 17481.631,E2 17481.631} C_VEL
LIN {X 0,Y 506.824,Z 574.517,A -85,B 0,C 180,E1 17479.266,E2 17479.266} C_VEL
LIN {X 0,Y 500.811,Z 564.934,A -85,B 0,C 180,E1 17476.768,E2 17476.768} C_VEL
LIN {X 0,Y 497.283,Z 559.403,A -85,B 0,C 180,E1 17475.093,E2 17475.093} C_VEL
LIN {X 0,Y 493.253,Z 553.909,A -85,B 0,C 180,E1 17472.944,E2 17472.944} C_VEL
LIN {X 0,Y 490.096,Z 549.424,A -85,B 0,C 180,E1 17470.938,E2 17470.938} C_VEL
LIN {X 0,Y 487.071,Z 545.628,A -85,B 0,C 180,E1 17468.619,E2 17468.619} C_VEL
LIN {X 0,Y 486.242,Z 543.976,A -85,B 0,C 180,E1 17467.8,E2 17467.8} C_VEL
LIN {X 0,Y 483.153,Z 540.488,A -85,B 0,C 180,E1 17463.916,E2 17463.916} C_VEL
LIN {X 0,Y 482.503,Z 538.143,A -85,B 0,C 180,E1 17461.9,E2 17461.9} C_VEL
LIN {X 0,Y 482.631,Z 538.362,A -85,B 0,C 180,E1 17457.15,E2 17457.15} C_VEL
LIN {X 0,Y 483.817,Z 541.648,A -85,B 0,C 180,E1 17454.426,E2 17454.426} C_VEL
LIN {X 0,Y 486.448,Z 544.317,A -85,B 0,C 180,E1 17451.489,E2 17451.489} C_VEL
LIN {X 0,Y 489.046,Z 548.386,A -85,B 0,C 180,E1 17449.277,E2 17449.277} C_VEL
LIN {X 0,Y 490.645,Z 550.183,A -85,B 0,C 180,E1 17448.182,E2 17448.182} C_VEL
LIN {X 0,Y 494.723,Z 555.901,A -85,B 0,C 180,E1 17445.725,E2 17445.725} C_VEL
LIN {X 0,Y 498.735,Z 561.443,A -85,B 0,C 180,E1 17443.699,E2 17443.699} C_VEL
LIN {X 0,Y 502.728,Z 567.135,A -85,B 0,C 180,E1 17441.924,E2 17441.924} C_VEL
LIN {X 0,Y 508.078,Z 574.795,A -85,B 0,C 180,E1 17439.821,E2 17439.821} C_VEL
LIN {X 0,Y 516.298,Z 587.145,A -85,B 0,C 180,E1 17437.001,E2 17437.001} C_VEL
LIN {X 0,Y 518.526,Z 590.87,A -85,B 0,C 180,E1 17436.293,E2 17436.293} C_VEL
LIN {X 0,Y 503.341,Z 805.987,A -85,B 0,C 180,E1 17432.946,E2 17432.946} C_VEL
LIN {X 0,Y 497.876,Z 882.767,A -85,B 0,C 180,E1 17431.733,E2 17431.733} C_VEL
LIN {X 0,Y 494.542,Z 910.883,A -85,B 0,C 180,E1 17431.18,E2 17431.18} C_VEL
LIN {X 0,Y 490.454,Z 935.638,A -85,B 0,C 180,E1 17430.525,E2 17430.525} C_VEL
LIN {X 0,Y 486.232,Z 956.817,A -85,B 0,C 180,E1 17429.834,E2 17429.834} C_VEL
LIN {X 0,Y 481.521,Z 977.259,A -85,B 0,C 180,E1 17429.032,E2 17429.032} C_VEL
LIN {X 0,Y 475.564,Z 999.905,A -85,B 0,C 180,E1 17427.983,E2 17427.983} C_VEL
LIN {X 0,Y 467.812,Z 1025.669,A -85,B 0,C 180,E1 17426.534,E2 17426.534} C_VEL
LIN {X 0,Y 461.207,Z 1045.239,A -85,B 0,C 180,E1 17425.237,E2 17425.237} C_VEL
LIN {X 0,Y 454.467,Z 1063.69,A -85,B 0,C 180,E1 17423.833,E2 17423.833} C_VEL
LIN {X 0,Y 447.3,Z 1082.059,A -85,B 0,C 180,E1 17422.229,E2 17422.229} C_VEL
LIN {X 0,Y 438.551,Z 1103.256,A -85,B 0,C 180,E1 17420.091,E2 17420.091} C_VEL
LIN {X 0,Y 429.708,Z 1123.078,A -85,B 0,C 180,E1 17417.715,E2 17417.715} C_VEL
LIN {X 0,Y 422.622,Z 1138.477,A -85,B 0,C 180,E1 17415.591,E2 17415.591} C_VEL
LIN {X 0,Y 415.673,Z 1153.254,A -85,B 0,C 180,E1 17413.268,E2 17413.268} C_VEL
LIN {X 0,Y 407.925,Z 1169.626,A -85,B 0,C 180,E1 17410.312,E2 17410.312} C_VEL
LIN {X 0,Y 400.414,Z 1185.297,A -85,B 0,C 180,E1 17406.957,E2 17406.957} C_VEL
LIN {X 0,Y 394.862,Z 1197.128,A -85,B 0,C 180,E1 17404.02,E2 17404.02} C_VEL
LIN {X 0,Y 390.121,Z 1207.72,A -85,B 0,C 180,E1 17400.999,E2 17400.999} C_VEL
LIN {X 0,Y 385.505,Z 1218.85,A -85,B 0,C 180,E1 17397.319,E2 17397.319} C_VEL
LIN {X 0,Y 381.688,Z 1228.862,A -85,B 0,C 180,E1 17393.292,E2 17393.292} C_VEL
LIN {X 0,Y 379.357,Z 1235.97,A -85,B 0,C 180,E1 17389.869,E2 17389.869} C_VEL
LIN {X 0,Y 377.836,Z 1241.627,A -85,B 0,C 180,E1 17386.599,E2 17386.599} C_VEL
LIN {X 0,Y 376.786,Z 1246.515,A -85,B 0,C 180,E1 17383.112,E2 17383.112} C_VEL
LIN {X 0,Y 376.19,Z 1250.834,A -85,B 0,C 180,E1 17379.015,E2 17379.015} C_VEL
LIN {X 0,Y 375.991,Z 1253.31,A -85,B 0,C 180,E1 17375.18,E2 17375.18} C_VEL
LIN {X 0,Y 375.952,Z 1254.387,A -85,B 0,C 180,E1 17371.974,E2 17371.974} C_VEL
LIN {X 0,Y 375.919,Z 1254.53,A -85,B 0,C 180,E1 17368.926,E2 17368.926} C_VEL
LIN {X 0,Y 375.975,Z 1253.767,A -85,B 0,C 180,E1 17365.791,E2 17365.791} C_VEL
LIN {X 0,Y 376.072,Z 1252.068,A -85,B 0,C 180,E1 17362.625,E2 17362.625} C_VEL
LIN {X 0,Y 376.328,Z 1249.41,A -85,B 0,C 180,E1 17359.43,E2 17359.43} C_VEL
LIN {X 0,Y 376.708,Z 1247.051,A -85,B 0,C 180,E1 17357.209,E2 17357.209} C_VEL
LIN {X 0,Y 375.958,Z 1245.678,A -85,B 0,C 180,E1 17356.053,E2 17356.053} C_VEL
LIN {X 0,Y 370.637,Z 1241.72,A -85,B 0,C 180,E1 17352.857,E2 17352.857} C_VEL
LIN {X 0,Y 370.415,Z 1240.334,A -85,B 0,C 180,E1 17351.933,E2 17351.933} C_VEL
LIN {X 0,Y 373.049,Z 1232.054,A -85,B 0,C 180,E1 17347.457,E2 17347.457} C_VEL
LIN {X 0,Y 376.016,Z 1224.117,A -85,B 0,C 180,E1 17343.969,E2 17343.969} C_VEL
LIN {X 0,Y 379.516,Z 1215.754,A -85,B 0,C 180,E1 17340.824,E2 17340.824} C_VEL
LIN {X 0,Y 383.834,Z 1206.213,A -85,B 0,C 180,E1 17337.716,E2 17337.716} C_VEL
LIN {X 0,Y 390.014,Z 1193.375,A -85,B 0,C 180,E1 17334.11,E2 17334.11} C_VEL
LIN {X 0,Y 397.397,Z 1178.294,A -85,B 0,C 180,E1 17330.574,E2 17330.574} C_VEL
LIN {X 0,Y 404.044,Z 1164.942,A -85,B 0,C 180,E1 17327.877,E2 17327.877} C_VEL
LIN {X 0,Y 410.752,Z 1151.403,A -85,B 0,C 180,E1 17325.481,E2 17325.481} C_VEL
LIN {X 0,Y 419.152,Z 1134.238,A -85,B 0,C 180,E1 17322.834,E2 17322.834} C_VEL
LIN {X 0,Y 428.646,Z 1113.881,A -85,B 0,C 180,E1 17320.181,E2 17320.181} C_VEL
LIN {X 0,Y 436.241,Z 1096.831,A -85,B 0,C 180,E1 17318.271,E2 17318.271} C_VEL
LIN {X 0,Y 443.432,Z 1079.831,A -85,B 0,C 180,E1 17316.602,E2 17316.602} C_VEL
LIN {X 0,Y 450.953,Z 1060.935,A -85,B 0,C 180,E1 17314.981,E2 17314.981} C_VEL
LIN {X 0,Y 459.986,Z 1036.245,A -85,B 0,C 180,E1 17313.182,E2 17313.182} C_VEL
LIN {X 0,Y 466.923,Z 1015.013,A -85,B 0,C 180,E1 17311.883,E2 17311.883} C_VEL
LIN {X 0,Y 472.826,Z 995.095,A -85,B 0,C 180,E1 17310.838,E2 17310.838} C_VEL
LIN {X 0,Y 478.218,Z 974.706,A -85,B 0,C 180,E1 17309.922,E2 17309.922} C_VEL
LIN {X 0,Y 483.299,Z 952.767,A -85,B 0,C 180,E1 17309.091,E2 17309.091} C_VEL
LIN {X 0,Y 488.765,Z 924.05,A -85,B 0,C 180,E1 17308.222,E2 17308.222} C_VEL
LIN {X 0,Y 492.175,Z 901.003,A -85,B 0,C 180,E1 17307.688,E2 17307.688} C_VEL
LIN {X 0,Y 494.616,Z 878.825,A -85,B 0,C 180,E1 17307.282,E2 17307.282} C_VEL
LIN {X 0,Y 510.082,Z 664.061,A -85,B 0,C 180,E1 17303.928,E2 17303.928} C_VEL
LIN {X 0,Y 515.072,Z 595.667,A -85,B 0,C 180,E1 17302.846,E2 17302.846} C_VEL
LIN {X 0,Y 507.786,Z 584.421,A -85,B 0,C 180,E1 17300.338,E2 17300.338} C_VEL
LIN {X 0,Y 501.953,Z 575.807,A -85,B 0,C 180,E1 17298.045,E2 17298.045} C_VEL
LIN {X 0,Y 497.844,Z 569.902,A -85,B 0,C 180,E1 17296.211,E2 17296.211} C_VEL
LIN {X 0,Y 495.236,Z 566.203,A -85,B 0,C 180,E1 17294.917,E2 17294.917} C_VEL
LIN {X 0,Y 492.165,Z 561.822,A -85,B 0,C 180,E1 17293.212,E2 17293.212} C_VEL
LIN {X 0,Y 488.729,Z 556.996,A -85,B 0,C 180,E1 17290.969,E2 17290.969} C_VEL
LIN {X 0,Y 485.689,Z 552.767,A -85,B 0,C 180,E1 17288.465,E2 17288.465} C_VEL
LIN {X 0,Y 485.055,Z 551.737,A -85,B 0,C 180,E1 17287.82,E2 17287.82} C_VEL
LIN {X 0,Y 482.13,Z 547.982,A -85,B 0,C 180,E1 17283.686,E2 17283.686} C_VEL
LIN {X 0,Y 481.717,Z 546.086,A -85,B 0,C 180,E1 17282.022,E2 17282.022} C_VEL
LIN {X 0,Y 481.78,Z 546.265,A -85,B 0,C 180,E1 17278.097,E2 17278.097} C_VEL
LIN {X 0,Y 483.508,Z 550.429,A -85,B 0,C 180,E1 17274.303,E2 17274.303} C_VEL
LIN {X 0,Y 485.469,Z 552.246,A -85,B 0,C 180,E1 17272.187,E2 17272.187} C_VEL
LIN {X 0,Y 488.151,Z 556.465,A -85,B 0,C 180,E1 17269.854,E2 17269.854} C_VEL
LIN {X 0,Y 489.553,Z 558.098,A -85,B 0,C 180,E1 17268.871,E2 17268.871} C_VEL
LIN {X 0,Y 493.347,Z 563.504,A -85,B 0,C 180,E1 17266.522,E2 17266.522} C_VEL
LIN {X 0,Y 497.605,Z 569.56,A -85,B 0,C 180,E1 17264.32,E2 17264.32} C_VEL
LIN {X 0,Y 504.23,Z 580.494,A -85,B 0,C 180,E1 17261.382,E2 17261.382} C_VEL
LIN {X 0,Y 510.594,Z 591.391,A -85,B 0,C 180,E1 17258.97,E2 17258.97} C_VEL
LIN {X 0,Y 515.184,Z 599.681,A -85,B 0,C 180,E1 17257.399,E2 17257.399} C_VEL
LIN {X 0,Y 499.338,Z 819.298,A -85,B 0,C 180,E1 17253.982,E2 17253.982} C_VEL
LIN {X 0,Y 493.639,Z 897.935,A -85,B 0,C 180,E1 17252.736,E2 17252.736} C_VEL
LIN {X 0,Y 490.138,Z 926.405,A -85,B 0,C 180,E1 17252.192,E2 17252.192} C_VEL
LIN {X 0,Y 485.803,Z 951.307,A -85,B 0,C 180,E1 17251.572,E2 17251.572} C_VEL
LIN {X 0,Y 481.429,Z 972.304,A -85,B 0,C 180,E1 17250.922,E2 17250.922} C_VEL
LIN {X 0,Y 476.616,Z 992.408,A -85,B 0,C 180,E1 17250.172,E2 17250.172} C_VEL
LIN {X 0,Y 470.986,Z 1013.227,A -85,B 0,C 180,E1 17249.253,E2 17249.253} C_VEL
LIN {X 0,Y 463.259,Z 1038.732,A -85,B 0,C 180,E1 17247.91,E2 17247.91} C_VEL
LIN {X 0,Y 455.071,Z 1062.474,A -85,B 0,C 180,E1 17246.387,E2 17246.387} C_VEL
LIN {X 0,Y 448.101,Z 1081.24,A -85,B 0,C 180,E1 17244.982,E2 17244.982} C_VEL
LIN {X 0,Y 441.107,Z 1098.856,A -85,B 0,C 180,E1 17243.478,E2 17243.478} C_VEL
LIN {X 0,Y 433.101,Z 1117.962,A -85,B 0,C 180,E1 17241.608,E2 17241.608} C_VEL
LIN {X 0,Y 423.13,Z 1140.455,A -85,B 0,C 180,E1 17239.012,E2 17239.012} C_VEL
LIN {X 0,Y 415.587,Z 1156.781,A -85,B 0,C 180,E1 17236.809,E2 17236.809} C_VEL
LIN {X 0,Y 408.788,Z 1171.226,A -85,B 0,C 180,E1 17234.593,E2 17234.593} C_VEL
LIN {X 0,Y 402.165,Z 1185.154,A -85,B 0,C 180,E1 17232.173,E2 17232.173} C_VEL
LIN {X 0,Y 395.54,Z 1199.202,A -85,B 0,C 180,E1 17229.389,E2 17229.389} C_VEL
LIN {X 0,Y 387.719,Z 1216.052,A -85,B 0,C 180,E1 17225.474,E2 17225.474} C_VEL
LIN {X 0,Y 382.498,Z 1227.87,A -85,B 0,C 180,E1 17222.233,E2 17222.233} C_VEL
LIN {X 0,Y 378.362,Z 1237.824,A -85,B 0,C 180,E1 17219.101,E2 17219.101} C_VEL
LIN {X 0,Y 374.919,Z 1246.993,A -85,B 0,C 180,E1 17215.773,E2 17215.773} C_VEL
LIN {X 0,Y 371.664,Z 1256.976,A -85,B 0,C 180,E1 17211.468,E2 17211.468} C_VEL
LIN {X 0,Y 369.796,Z 1264.115,A -85,B 0,C 180,E1 17207.634,E2 17207.634} C_VEL
LIN {X 0,Y 368.773,Z 1269.205,A -85,B 0,C 180,E1 17204.291,E2 17204.291} C_VEL
LIN {X 0,Y 368.251,Z 1273.048,A -85,B 0,C 180,E1 17201.122,E2 17201.122} C_VEL
LIN {X 0,Y 367.997,Z 1275.925,A -85,B 0,C 180,E1 17197.972,E2 17197.972} C_VEL
LIN {X 0,Y 367.954,Z 1277.783,A -85,B 0,C 180,E1 17194.995,E2 17194.995} C_VEL
LIN {X 0,Y 367.95,Z 1278.818,A -85,B 0,C 180,E1 17191.876,E2 17191.876} C_VEL
LIN {X 0,Y 367.925,Z 1278.936,A -85,B 0,C 180,E1 17188.917,E2 17188.917} C_VEL
LIN {X 0,Y 367.951,Z 1278.141,A -85,B 0,C 180,E1 17185.798,E2 17185.798} C_VEL
LIN {X 0,Y 367.994,Z 1276.381,A -85,B 0,C 180,E1 17182.64,E2 17182.64} C_VEL
LIN {X 0,Y 368.193,Z 1273.555,A -85,B 0,C 180,E1 17179.366,E2 17179.366} C_VEL
LIN {X 0,Y 368.689,Z 1269.787,A -85,B 0,C 180,E1 17176.145,E2 17176.145} C_VEL
LIN {X 0,Y 369.607,Z 1264.921,A -85,B 0,C 180,E1 17172.858,E2 17172.858} C_VEL
LIN {X 0,Y 371.11,Z 1258.869,A -85,B 0,C 180,E1 17169.505,E2 17169.505} C_VEL
LIN {X 0,Y 373.506,Z 1251.107,A -85,B 0,C 180,E1 17165.906,E2 17165.906} C_VEL
LIN {X 0,Y 377.65,Z 1239.673,A -85,B 0,C 180,E1 17161.525,E2 17161.525} C_VEL
LIN {X 0,Y 382.023,Z 1228.957,A -85,B 0,C 180,E1 17158.092,E2 17158.092} C_VEL
LIN {X 0,Y 386.871,Z 1217.903,A -85,B 0,C 180,E1 17155.016,E2 17155.016} C_VEL
LIN {X 0,Y 392.807,Z 1204.933,A -85,B 0,C 180,E1 17151.865,E2 17151.865} C_VEL
LIN {X 0,Y 401.029,Z 1187.53,A -85,B 0,C 180,E1 17148.275,E2 17148.275} C_VEL
LIN {X 0,Y 407.933,Z 1172.966,A -85,B 0,C 180,E1 17145.7,E2 17145.7} C_VEL
LIN {X 0,Y 415.003,Z 1157.938,A -85,B 0,C 180,E1 17143.367,E2 17143.367} C_VEL
LIN {X 0,Y 422.166,Z 1142.433,A -85,B 0,C 180,E1 17141.25,E2 17141.25} C_VEL
LIN {X 0,Y 430.76,Z 1123.304,A -85,B 0,C 180,E1 17138.972,E2 17138.972} C_VEL
LIN {X 0,Y 440.231,Z 1100.88,A -85,B 0,C 180,E1 17136.716,E2 17136.716} C_VEL
LIN {X 0,Y 447.459,Z 1082.716,A -85,B 0,C 180,E1 17135.144,E2 17135.144} C_VEL
LIN {X 0,Y 454.402,Z 1064.1,A -85,B 0,C 180,E1 17133.734,E2 17133.734} C_VEL
LIN {X 0,Y 461.328,Z 1044.168,A -85,B 0,C 180,E1 17132.429,E2 17132.429} C_VEL
LIN {X 0,Y 469.141,Z 1019.583,A -85,B 0,C 180,E1 17131.058,E2 17131.058} C_VEL
LIN {X 0,Y 475.884,Z 994.957,A -85,B 0,C 180,E1 17129.938,E2 17129.938} C_VEL
LIN {X 0,Y 480.997,Z 973.815,A -85,B 0,C 180,E1 17129.136,E2 17129.136} C_VEL
LIN {X 0,Y 485.464,Z 952.554,A -85,B 0,C 180,E1 17128.47,E2 17128.47} C_VEL
LIN {X 0,Y 489.372,Z 930.429,A -85,B 0,C 180,E1 17127.907,E2 17127.907} C_VEL
LIN {X 0,Y 493.2,Z 901.751,A -85,B 0,C 180,E1 17127.334,E2 17127.334} C_VEL
LIN {X 0,Y 496.858,Z 853.477,A -85,B 0,C 180,E1 17126.558,E2 17126.558} C_VEL
LIN {X 0,Y 512.313,Z 636.709,A -85,B 0,C 180,E1 17123.18,E2 17123.18} C_VEL
LIN {X 0,Y 514.997,Z 599.332,A -85,B 0,C 180,E1 17122.578,E2 17122.578} C_VEL
LIN {X 0,Y 507.009,Z 585.339,A -85,B 0,C 180,E1 17119.769,E2 17119.769} C_VEL
LIN {X 0,Y 500.443,Z 574.35,A -85,B 0,C 180,E1 17117.08,E2 17117.08} C_VEL
LIN {X 0,Y 495.73,Z 566.958,A -85,B 0,C 180,E1 17114.842,E2 17114.842} C_VEL
LIN {X 0,Y 491.88,Z 561.599,A -85,B 0,C 180,E1 17112.742,E2 17112.742} C_VEL
LIN {X 0,Y 488.779,Z 557.158,A -85,B 0,C 180,E1 17110.729,E2 17110.729} C_VEL
LIN {X 0,Y 485.773,Z 553.194,A -85,B 0,C 180,E1 17108.344,E2 17108.344} C_VEL
LIN {X 0,Y 485.015,Z 551.789,A -85,B 0,C 180,E1 17107.582,E2 17107.582} C_VEL
LIN {X 0,Y 482.065,Z 548.218,A -85,B 0,C 180,E1 17103.687,E2 17103.687} C_VEL
LIN {X 0,Y 481.529,Z 546.084,A -85,B 0,C 180,E1 17101.904,E2 17101.904} C_VEL
LIN {X 0,Y 481.62,Z 546.251,A -85,B 0,C 180,E1 17097.263,E2 17097.263} C_VEL
LIN {X 0,Y 482.841,Z 549.636,A -85,B 0,C 180,E1 17094.415,E2 17094.415} C_VEL
LIN {X 0,Y 485.284,Z 552.14,A -85,B 0,C 180,E1 17091.648,E2 17091.648} C_VEL
LIN {X 0,Y 487.914,Z 556.271,A -85,B 0,C 180,E1 17089.372,E2 17089.372} C_VEL
LIN {X 0,Y 489.323,Z 557.88,A -85,B 0,C 180,E1 17088.388,E2 17088.388} C_VEL
LIN {X 0,Y 493.324,Z 563.61,A -85,B 0,C 180,E1 17085.923,E2 17085.923} C_VEL
LIN {X 0,Y 497.275,Z 569.167,A -85,B 0,C 180,E1 17083.89,E2 17083.89} C_VEL
LIN {X 0,Y 501.346,Z 575.057,A -85,B 0,C 180,E1 17082.053,E2 17082.053} C_VEL
LIN {X 0,Y 506.897,Z 583.256,A -85,B 0,C 180,E1 17079.844,E2 17079.844} C_VEL
LIN {X 0,Y 514.224,Z 594.435,A -85,B 0,C 180,E1 17077.296,E2 17077.296} C_VEL
LIN {X 0,Y 514.994,Z 596.003,A -85,B 0,C 180,E1 17077.034,E2 17077.034} C_VEL
LIN {X 0,Y 499.441,Z 810.687,A -85,B 0,C 180,E1 17073.695,E2 17073.695} C_VEL
LIN {X 0,Y 494.116,Z 883.266,A -85,B 0,C 180,E1 17072.547,E2 17072.547} C_VEL
LIN {X 0,Y 490.644,Z 911.679,A -85,B 0,C 180,E1 17071.987,E2 17071.987} C_VEL
LIN {X 0,Y 486.534,Z 936.021,A -85,B 0,C 180,E1 17071.345,E2 17071.345} C_VEL
LIN {X 0,Y 482.239,Z 957.091,A -85,B 0,C 180,E1 17070.661,E2 17070.661} C_VEL
LIN {X 0,Y 477.42,Z 977.533,A -85,B 0,C 180,E1 17069.863,E2 17069.863} C_VEL
LIN {X 0,Y 471.411,Z 999.864,A -85,B 0,C 180,E1 17068.833,E2 17068.833} C_VEL
LIN {X 0,Y 463.433,Z 1025.792,A -85,B 0,C 180,E1 17067.381,E2 17067.381} C_VEL
LIN {X 0,Y 456.603,Z 1045.513,A -85,B 0,C 180,E1 17066.078,E2 17066.078} C_VEL
LIN {X 0,Y 449.686,Z 1063.964,A -85,B 0,C 180,E1 17064.675,E2 17064.675} C_VEL
LIN {X 0,Y 442.496,Z 1081.914,A -85,B 0,C 180,E1 17063.108,E2 17063.108} C_VEL
LIN {X 0,Y 434.329,Z 1101.129,A -85,B 0,C 180,E1 17061.181,E2 17061.181} C_VEL
LIN {X 0,Y 424.666,Z 1122.353,A -85,B 0,C 180,E1 17058.672,E2 17058.672} C_VEL
LIN {X 0,Y 416.859,Z 1138.752,A -85,B 0,C 180,E1 17056.405,E2 17056.405} C_VEL
LIN {X 0,Y 409.657,Z 1153.53,A -85,B 0,C 180,E1 17054.065,E2 17054.065} C_VEL
LIN {X 0,Y 401.959,Z 1169.145,A -85,B 0,C 180,E1 17051.227,E2 17051.227} C_VEL
LIN {X 0,Y 393.827,Z 1185.462,A -85,B 0,C 180,E1 17047.714,E2 17047.714} C_VEL
LIN {X 0,Y 387.97,Z 1197.433,A -85,B 0,C 180,E1 17044.7,E2 17044.7} C_VEL
LIN {X 0,Y 382.999,Z 1207.995,A -85,B 0,C 180,E1 17041.641,E2 17041.641} C_VEL
LIN {X 0,Y 378.129,Z 1219.125,A -85,B 0,C 180,E1 17037.898,E2 17037.898} C_VEL
LIN {X 0,Y 374.095,Z 1229.136,A -85,B 0,C 180,E1 17033.794,E2 17033.794} C_VEL
LIN {X 0,Y 371.62,Z 1236.241,A -85,B 0,C 180,E1 17030.301,E2 17030.301} C_VEL
LIN {X 0,Y 369.972,Z 1241.966,A -85,B 0,C 180,E1 17026.917,E2 17026.917} C_VEL
LIN {X 0,Y 368.841,Z 1246.921,A -85,B 0,C 180,E1 17023.29,E2 17023.29} C_VEL
LIN {X 0,Y 368.201,Z 1251.208,A -85,B 0,C 180,E1 17019.054,E2 17019.054} C_VEL
LIN {X 0,Y 368,Z 1253.574,A -85,B 0,C 180,E1 17015.293,E2 17015.293} C_VEL
LIN {X 0,Y 367.956,Z 1254.65,A -85,B 0,C 180,E1 17012.017,E2 17012.017} C_VEL
LIN {X 0,Y 367.924,Z 1254.793,A -85,B 0,C 180,E1 17008.903,E2 17008.903} C_VEL
LIN {X 0,Y 367.981,Z 1254.044,A -85,B 0,C 180,E1 17005.735,E2 17005.735} C_VEL
LIN {X 0,Y 368.084,Z 1252.358,A -85,B 0,C 180,E1 17002.501,E2 17002.501} C_VEL
LIN {X 0,Y 368.381,Z 1249.674,A -85,B 0,C 180,E1 16999.199,E2 16999.199} C_VEL
LIN {X 0,Y 369.022,Z 1246.065,A -85,B 0,C 180,E1 16995.938,E2 16995.938} C_VEL
LIN {X 0,Y 370.142,Z 1241.281,A -85,B 0,C 180,E1 16992.545,E2 16992.545} C_VEL
LIN {X 0,Y 370.415,Z 1240.334,A -85,B 0,C 180,E1 16991.933,E2 16991.933} C_VEL
LIN {X 0,Y 370.015,Z 1238.568,A -85,B 0,C 180,E1 16990.766,E2 16990.766} C_VEL
LIN {X 0,Y 365.658,Z 1233.433,A -85,B 0,C 180,E1 16987.532,E2 16987.532} C_VEL
LIN {X 0,Y 365.701,Z 1231.593,A -85,B 0,C 180,E1 16986.615,E2 16986.615} C_VEL
LIN {X 0,Y 368.747,Z 1223.993,A -85,B 0,C 180,E1 16983.242,E2 16983.242} C_VEL
LIN {X 0,Y 372.472,Z 1215.578,A -85,B 0,C 180,E1 16980.039,E2 16980.039} C_VEL
LIN {X 0,Y 377.32,Z 1205.479,A -85,B 0,C 180,E1 16976.727,E2 16976.727} C_VEL
LIN {X 0,Y 384.605,Z 1190.98,A -85,B 0,C 180,E1 16972.706,E2 16972.706} C_VEL
LIN {X 0,Y 391.218,Z 1178.136,A -85,B 0,C 180,E1 16969.706,E2 16969.706} C_VEL
LIN {X 0,Y 397.902,Z 1165.213,A -85,B 0,C 180,E1 16967.073,E2 16967.073} C_VEL
LIN {X 0,Y 404.868,Z 1151.673,A -85,B 0,C 180,E1 16964.656,E2 16964.656} C_VEL
LIN {X 0,Y 413.221,Z 1135.162,A -85,B 0,C 180,E1 16962.088,E2 16962.088} C_VEL
LIN {X 0,Y 423.108,Z 1114.697,A -85,B 0,C 180,E1 16959.391,E2 16959.391} C_VEL
LIN {X 0,Y 430.922,Z 1097.698,A -85,B 0,C 180,E1 16957.475,E2 16957.475} C_VEL
LIN {X 0,Y 438.311,Z 1080.756,A -85,B 0,C 180,E1 16955.803,E2 16955.803} C_VEL
LIN {X 0,Y 446.023,Z 1061.926,A -85,B 0,C 180,E1 16954.18,E2 16954.18} C_VEL
LIN {X 0,Y 454.979,Z 1038.292,A -85,B 0,C 180,E1 16952.44,E2 16952.44} C_VEL
LIN {X 0,Y 462.688,Z 1015.273,A -85,B 0,C 180,E1 16951.03,E2 16951.03} C_VEL
LIN {X 0,Y 468.731,Z 995.352,A -85,B 0,C 180,E1 16949.989,E2 16949.989} C_VEL
LIN {X 0,Y 474.245,Z 974.962,A -85,B 0,C 180,E1 16949.077,E2 16949.077} C_VEL
LIN {X 0,Y 479.502,Z 952.75,A -85,B 0,C 180,E1 16948.241,E2 16948.241} C_VEL
LIN {X 0,Y 485.082,Z 923.935,A -85,B 0,C 180,E1 16947.378,E2 16947.378} C_VEL
LIN {X 0,Y 488.524,Z 901.087,A -85,B 0,C 180,E1 16946.853,E2 16946.853} C_VEL
LIN {X 0,Y 491.016,Z 878.851,A -85,B 0,C 180,E1 16946.448,E2 16946.448} C_VEL
LIN {X 0,Y 506.924,Z 663.771,A -85,B 0,C 180,E1 16943.092,E2 16943.092} C_VEL
LIN {X 0,Y 511.669,Z 600.778,A -85,B 0,C 180,E1 16942.103,E2 16942.103} C_VEL
LIN {X 0,Y 503.8,Z 588.463,A -85,B 0,C 180,E1 16939.236,E2 16939.236} C_VEL
LIN {X 0,Y 497.252,Z 578.809,A -85,B 0,C 180,E1 16936.429,E2 16936.429} C_VEL
LIN {X 0,Y 493.71,Z 573.754,A -85,B 0,C 180,E1 16934.665,E2 16934.665} C_VEL
LIN {X 0,Y 490.701,Z 569.406,A -85,B 0,C 180,E1 16932.953,E2 16932.953} C_VEL
LIN {X 0,Y 487.593,Z 564.876,A -85,B 0,C 180,E1 16930.875,E2 16930.875} C_VEL
LIN {X 0,Y 484.527,Z 560.579,A -85,B 0,C 180,E1 16928.306,E2 16928.306} C_VEL
LIN {X 0,Y 483.964,Z 559.623,A -85,B 0,C 180,E1 16927.718,E2 16927.718} C_VEL
LIN {X 0,Y 481.105,Z 555.861,A -85,B 0,C 180,E1 16923.575,E2 16923.575} C_VEL
LIN {X 0,Y 480.712,Z 554.021,A -85,B 0,C 180,E1 16921.907,E2 16921.907} C_VEL
LIN {X 0,Y 480.794,Z 554.299,A -85,B 0,C 180,E1 16918.093,E2 16918.093} C_VEL
LIN {X 0,Y 482.533,Z 558.409,A -85,B 0,C 180,E1 16914.292,E2 16914.292} C_VEL
LIN {X 0,Y 484.363,Z 560.193,A -85,B 0,C 180,E1 16912.289,E2 16912.289} C_VEL
LIN {X 0,Y 487.019,Z 564.348,A -85,B 0,C 180,E1 16909.95,E2 16909.95} C_VEL
LIN {X 0,Y 488.316,Z 565.937,A -85,B 0,C 180,E1 16909.022,E2 16909.022} C_VEL
LIN {X 0,Y 491.956,Z 571.211,A -85,B 0,C 180,E1 16906.722,E2 16906.722} C_VEL
LIN {X 0,Y 496.032,Z 577.109,A -85,B 0,C 180,E1 16904.569,E2 16904.569} C_VEL
LIN {X 0,Y 502.61,Z 588.205,A -85,B 0,C 180,E1 16901.59,E2 16901.59} C_VEL
LIN {X 0,Y 508.736,Z 598.949,A -85,B 0,C 180,E1 16899.221,E2 16899.221} C_VEL
LIN {X 0,Y 511.741,Z 604.641,A -85,B 0,C 180,E1 16898.152,E2 16898.152} C_VEL
LIN {X 0,Y 495.558,Z 823.242,A -85,B 0,C 180,E1 16894.753,E2 16894.753} C_VEL
LIN {X 0,Y 489.987,Z 897.861,A -85,B 0,C 180,E1 16893.57,E2 16893.57} C_VEL
LIN {X 0,Y 486.344,Z 926.676,A -85,B 0,C 180,E1 16893.019,E2 16893.019} C_VEL
LIN {X 0,Y 481.989,Z 951.161,A -85,B 0,C 180,E1 16892.413,E2 16892.413} C_VEL
LIN {X 0,Y 477.535,Z 972.082,A -85,B 0,C 180,E1 16891.77,E2 16891.77} C_VEL
LIN {X 0,Y 472.557,Z 992.407,A -85,B 0,C 180,E1 16891.017,E2 16891.017} C_VEL
LIN {X 0,Y 466.809,Z 1013.164,A -85,B 0,C 180,E1 16890.105,E2 16890.105} C_VEL
LIN {X 0,Y 459.127,Z 1037.978,A -85,B 0,C 180,E1 16888.807,E2 16888.807} C_VEL
LIN {X 0,Y 450.871,Z 1061.39,A -85,B 0,C 180,E1 16887.316,E2 16887.316} C_VEL
LIN {X 0,Y 443.651,Z 1080.345,A -85,B 0,C 180,E1 16885.908,E2 16885.908} C_VEL
LIN {X 0,Y 436.485,Z 1097.912,A -85,B 0,C 180,E1 16884.418,E2 16884.418} C_VEL
LIN {X 0,Y 428.503,Z 1116.421,A -85,B 0,C 180,E1 16882.618,E2 16882.618} C_VEL
LIN {X 0,Y 418.461,Z 1138.546,A -85,B 0,C 180,E1 16880.092,E2 16880.092} C_VEL
LIN {X 0,Y 409.92,Z 1156.4,A -85,B 0,C 180,E1 16877.683,E2 16877.683} C_VEL
LIN {X 0,Y 402.504,Z 1171.595,A -85,B 0,C 180,E1 16875.33,E2 16875.33} C_VEL
LIN {X 0,Y 395.558,Z 1185.662,A -85,B 0,C 180,E1 16872.848,E2 16872.848} C_VEL
LIN {X 0,Y 387.564,Z 1202.046,A -85,B 0,C 180,E1 16869.52,E2 16869.52} C_VEL
LIN {X 0,Y 380.297,Z 1216.947,A -85,B 0,C 180,E1 16865.902,E2 16865.902} C_VEL
LIN {X 0,Y 375.149,Z 1228.121,A -85,B 0,C 180,E1 16862.762,E2 16862.762} C_VEL
LIN {X 0,Y 370.84,Z 1238.019,A -85,B 0,C 180,E1 16859.572,E2 16859.572} C_VEL
LIN {X 0,Y 366.798,Z 1248.382,A -85,B 0,C 180,E1 16855.692,E2 16855.692} C_VEL
LIN {X 0,Y 363.63,Z 1257.641,A -85,B 0,C 180,E1 16851.458,E2 16851.458} C_VEL
LIN {X 0,Y 361.878,Z 1264.108,A -85,B 0,C 180,E1 16847.867,E2 16847.867} C_VEL
LIN {X 0,Y 360.833,Z 1268.936,A -85,B 0,C 180,E1 16844.612,E2 16844.612} C_VEL
LIN {X 0,Y 360.274,Z 1272.781,A -85,B 0,C 180,E1 16841.371,E2 16841.371} C_VEL
LIN {X 0,Y 360.008,Z 1275.66,A -85,B 0,C 180,E1 16838.15,E2 16838.15} C_VEL
LIN {X 0,Y 359.957,Z 1277.52,A -85,B 0,C 180,E1 16835.107,E2 16835.107} C_VEL
LIN {X 0,Y 359.955,Z 1278.531,A -85,B 0,C 180,E1 16832.077,E2 16832.077} C_VEL
LIN {X 0,Y 359.93,Z 1278.674,A -85,B 0,C 180,E1 16828.893,E2 16828.893} C_VEL
LIN {X 0,Y 359.953,Z 1277.878,A -85,B 0,C 180,E1 16825.706,E2 16825.706} C_VEL
LIN {X 0,Y 359.992,Z 1276.14,A -85,B 0,C 180,E1 16822.507,E2 16822.507} C_VEL
LIN {X 0,Y 360.221,Z 1273.288,A -85,B 0,C 180,E1 16819.128,E2 16819.128} C_VEL
LIN {X 0,Y 360.737,Z 1269.592,A -85,B 0,C 180,E1 16815.89,E2 16815.89} C_VEL
LIN {X 0,Y 361.739,Z 1264.649,A -85,B 0,C 180,E1 16812.474,E2 16812.474} C_VEL
LIN {X 0,Y 363.335,Z 1258.595,A -85,B 0,C 180,E1 16809.046,E2 16809.046} C_VEL
LIN {X 0,Y 365.737,Z 1251.253,A -85,B 0,C 180,E1 16805.56,E2 16805.56} C_VEL
LIN {X 0,Y 369.889,Z 1240.396,A -85,B 0,C 180,E1 16801.248,E2 16801.248} C_VEL
LIN {X 0,Y 374.659,Z 1229.205,A -85,B 0,C 180,E1 16797.57,E2 16797.57} C_VEL
LIN {X 0,Y 379.72,Z 1218.148,A -85,B 0,C 180,E1 16794.424,E2 16794.424} C_VEL
LIN {X 0,Y 385.655,Z 1205.723,A -85,B 0,C 180,E1 16791.341,E2 16791.341} C_VEL
LIN {X 0,Y 393.74,Z 1189.399,A -85,B 0,C 180,E1 16787.862,E2 16787.862} C_VEL
LIN {X 0,Y 401.937,Z 1172.687,A -85,B 0,C 180,E1 16784.86,E2 16784.86} C_VEL
LIN {X 0,Y 409.136,Z 1157.933,A -85,B 0,C 180,E1 16782.55,E2 16782.55} C_VEL
LIN {X 0,Y 416.436,Z 1142.668,A -85,B 0,C 180,E1 16780.449,E2 16780.449} C_VEL
LIN {X 0,Y 424.499,Z 1125.274,A -85,B 0,C 180,E1 16778.352,E2 16778.352} C_VEL
LIN {X 0,Y 434.753,Z 1101.953,A -85,B 0,C 180,E1 16775.961,E2 16775.961} C_VEL
LIN {X 0,Y 442.747,Z 1082.44,A -85,B 0,C 180,E1 16774.268,E2 16774.268} C_VEL
LIN {X 0,Y 449.877,Z 1063.825,A -85,B 0,C 180,E1 16772.861,E2 16772.861} C_VEL
LIN {X 0,Y 456.973,Z 1043.892,A -85,B 0,C 180,E1 16771.559,E2 16771.559} C_VEL
LIN {X 0,Y 464.976,Z 1019.308,A -85,B 0,C 180,E1 16770.195,E2 16770.195} C_VEL
LIN {X 0,Y 471.877,Z 994.683,A -85,B 0,C 180,E1 16769.082,E2 16769.082} C_VEL
LIN {X 0,Y 477.106,Z 973.523,A -85,B 0,C 180,E1 16768.285,E2 16768.285} C_VEL
LIN {X 0,Y 481.753,Z 951.843,A -85,B 0,C 180,E1 16767.613,E2 16767.613} C_VEL
LIN {X 0,Y 485.828,Z 929.106,A -85,B 0,C 180,E1 16767.043,E2 16767.043} C_VEL
LIN {X 0,Y 489.805,Z 898.683,A -85,B 0,C 180,E1 16766.45,E2 16766.45} C_VEL
LIN {X 0,Y 494.58,Z 835.343,A -85,B 0,C 180,E1 16765.443,E2 16765.443} C_VEL
LIN {X 0,Y 510.393,Z 620.578,A -85,B 0,C 180,E1 16762.1,E2 16762.1} C_VEL
LIN {X 0,Y 511.585,Z 604.234,A -85,B 0,C 180,E1 16761.832,E2 16761.832} C_VEL
LIN {X 0,Y 504.434,Z 591.538,A -85,B 0,C 180,E1 16759.211,E2 16759.211} C_VEL
LIN {X 0,Y 498.566,Z 581.534,A -85,B 0,C 180,E1 16756.726,E2 16756.726} C_VEL
LIN {X 0,Y 494.188,Z 574.513,A -85,B 0,C 180,E1 16754.59,E2 16754.59} C_VEL
LIN {X 0,Y 490.415,Z 569.175,A -85,B 0,C 180,E1 16752.481,E2 16752.481} C_VEL
LIN {X 0,Y 487.468,Z 564.888,A -85,B 0,C 180,E1 16750.519,E2 16750.519} C_VEL
LIN {X 0,Y 484.544,Z 560.881,A -85,B 0,C 180,E1 16748.126,E2 16748.126} C_VEL
LIN {X 0,Y 483.796,Z 559.596,A -85,B 0,C 180,E1 16747.362,E2 16747.362} C_VEL
LIN {X 0,Y 481.032,Z 556.098,A -85,B 0,C 180,E1 16743.575,E2 16743.575} C_VEL
LIN {X 0,Y 480.519,Z 554.018,A -85,B 0,C 180,E1 16741.789,E2 16741.789} C_VEL
LIN {X 0,Y 480.61,Z 554.141,A -85,B 0,C 180,E1 16737.377,E2 16737.377} C_VEL
LIN {X 0,Y 481.786,Z 557.515,A -85,B 0,C 180,E1 16734.522,E2 16734.522} C_VEL
LIN {X 0,Y 484.178,Z 560.092,A -85,B 0,C 180,E1 16731.748,E2 16731.748} C_VEL
LIN {X 0,Y 486.943,Z 564.32,A -85,B 0,C 180,E1 16729.35,E2 16729.35} C_VEL
LIN {X 0,Y 488.165,Z 565.875,A -85,B 0,C 180,E1 16728.48,E2 16728.48} C_VEL
LIN {X 0,Y 491.931,Z 571.317,A -85,B 0,C 180,E1 16726.123,E2 16726.123} C_VEL
LIN {X 0,Y 495.707,Z 576.713,A -85,B 0,C 180,E1 16724.138,E2 16724.138} C_VEL
LIN {X 0,Y 501.02,Z 584.408,A -85,B 0,C 180,E1 16721.74,E2 16721.74} C_VEL
LIN {X 0,Y 507.754,Z 594.834,A -85,B 0,C 180,E1 16719.119,E2 16719.119} C_VEL
LIN {X 0,Y 511.567,Z 600.909,A -85,B 0,C 180,E1 16717.788,E2 16717.788} C_VEL
LIN {X 0,Y 495.579,Z 816.049,A -85,B 0,C 180,E1 16714.445,E2 16714.445} C_VEL
LIN {X 0,Y 490.448,Z 883.872,A -85,B 0,C 180,E1 16713.371,E2 16713.371} C_VEL
LIN {X 0,Y 486.76,Z 912.995,A -85,B 0,C 180,E1 16712.795,E2 16712.795} C_VEL
LIN {X 0,Y 482.672,Z 936.62,A -85,B 0,C 180,E1 16712.171,E2 16712.171} C_VEL
LIN {X 0,Y 478.348,Z 957.365,A -85,B 0,C 180,E1 16711.501,E2 16711.501} C_VEL
LIN {X 0,Y 473.42,Z 977.806,A -85,B 0,C 180,E1 16710.707,E2 16710.707} C_VEL
LIN {X 0,Y 467.152,Z 1000.579,A -85,B 0,C 180,E1 16709.66,E2 16709.66} C_VEL
LIN {X 0,Y 459.134,Z 1025.975,A -85,B 0,C 180,E1 16708.241,E2 16708.241} C_VEL
LIN {X 0,Y 451.879,Z 1046.384,A -85,B 0,C 180,E1 16706.893,E2 16706.893} C_VEL
LIN {X 0,Y 444.826,Z 1064.694,A -85,B 0,C 180,E1 16705.497,E2 16705.497} C_VEL
LIN {X 0,Y 437.236,Z 1083.104,A -85,B 0,C 180,E1 16703.882,E2 16703.882} C_VEL
LIN {X 0,Y 427.903,Z 1104.371,A -85,B 0,C 180,E1 16701.719,E2 16701.719} C_VEL
LIN {X 0,Y 418.511,Z 1124.128,A -85,B 0,C 180,E1 16699.324,E2 16699.324} C_VEL
LIN {X 0,Y 411.189,Z 1139.028,A -85,B 0,C 180,E1 16697.241,E2 16697.241} C_VEL
LIN {X 0,Y 403.81,Z 1153.642,A -85,B 0,C 180,E1 16694.913,E2 16694.913} C_VEL
LIN {X 0,Y 395.729,Z 1169.421,A -85,B 0,C 180,E1 16692.022,E2 16692.022} C_VEL
LIN {X 0,Y 387.251,Z 1185.739,A -85,B 0,C 180,E1 16688.47,E2 16688.47} C_VEL
LIN {X 0,Y 381.163,Z 1197.679,A -85,B 0,C 180,E1 16685.421,E2 16685.421} C_VEL
LIN {X 0,Y 375.928,Z 1208.271,A -85,B 0,C 180,E1 16682.308,E2 16682.308} C_VEL
LIN {X 0,Y 370.746,Z 1219.531,A -85,B 0,C 180,E1 16678.452,E2 16678.452} C_VEL
LIN {X 0,Y 366.53,Z 1229.409,A -85,B 0,C 180,E1 16674.317,E2 16674.317} C_VEL
LIN {X 0,Y 363.992,Z 1236.219,A -85,B 0,C 180,E1 16670.914,E2 16670.914} C_VEL
LIN {X 0,Y 362.22,Z 1241.921,A -85,B 0,C 180,E1 16667.502,E2 16667.502} C_VEL
LIN {X 0,Y 361.063,Z 1246.559,A -85,B 0,C 180,E1 16664.097,E2 16664.097} C_VEL
LIN {X 0,Y 360.389,Z 1250.17,A -85,B 0,C 180,E1 16660.705,E2 16660.705} C_VEL
LIN {X 0,Y 360.07,Z 1253.114,A -85,B 0,C 180,E1 16656.85,E2 16656.85} C_VEL
LIN {X 0,Y 359.966,Z 1254.827,A -85,B 0,C 180,E1 16652.699,E2 16652.699} C_VEL
LIN {X 0,Y 359.923,Z 1255.077,A -85,B 0,C 180,E1 16649.038,E2 16649.038} C_VEL
LIN {X 0,Y 359.987,Z 1254.322,A -85,B 0,C 180,E1 16645.676,E2 16645.676} C_VEL
LIN {X 0,Y 360.092,Z 1252.694,A -85,B 0,C 180,E1 16642.441,E2 16642.441} C_VEL
LIN {X 0,Y 360.433,Z 1249.939,A -85,B 0,C 180,E1 16638.958,E2 16638.958} C_VEL
LIN {X 0,Y 361.089,Z 1246.458,A -85,B 0,C 180,E1 16635.726,E2 16635.726} C_VEL
LIN {X 0,Y 362.252,Z 1241.796,A -85,B 0,C 180,E1 16632.318,E2 16632.318} C_VEL
LIN {X 0,Y 364.048,Z 1236.07,A -85,B 0,C 180,E1 16628.906,E2 16628.906} C_VEL
LIN {X 0,Y 365.701,Z 1231.593,A -85,B 0,C 180,E1 16626.615,E2 16626.615} C_VEL
LIN {X 0,Y 365.655,Z 1229.313,A -85,B 0,C 180,E1 16625.455,E2 16625.455} C_VEL
LIN {X 0,Y 362.5,Z 1223.248,A -85,B 0,C 180,E1 16622.286,E2 16622.286} C_VEL
LIN {X 0,Y 362.896,Z 1220.993,A -85,B 0,C 180,E1 16621.294,E2 16621.294} C_VEL
LIN {X 0,Y 368.558,Z 1209.274,A -85,B 0,C 180,E1 16617.133,E2 16617.133} C_VEL
LIN {X 0,Y 373.994,Z 1198.763,A -85,B 0,C 180,E1 16613.966,E2 16613.966} C_VEL
LIN {X 0,Y 379.956,Z 1187.534,A -85,B 0,C 180,E1 16611.021,E2 16611.021} C_VEL
LIN {X 0,Y 386.884,Z 1174.72,A -85,B 0,C 180,E1 16608.102,E2 16608.102} C_VEL
LIN {X 0,Y 396.442,Z 1156.936,A -85,B 0,C 180,E1 16604.658,E2 16604.658} C_VEL
LIN {X 0,Y 404.516,Z 1141.514,A -85,B 0,C 180,E1 16602.131,E2 16602.131} C_VEL
LIN {X 0,Y 412.471,Z 1125.904,A -85,B 0,C 180,E1 16599.905,E2 16599.905} C_VEL
LIN {X 0,Y 420.72,Z 1109.09,A -85,B 0,C 180,E1 16597.819,E2 16597.819} C_VEL
LIN {X 0,Y 430.705,Z 1087.628,A -85,B 0,C 180,E1 16595.536,E2 16595.536} C_VEL
LIN {X 0,Y 439.686,Z 1066.556,A -85,B 0,C 180,E1 16593.657,E2 16593.657} C_VEL
LIN {X 0,Y 446.938,Z 1048.308,A -85,B 0,C 180,E1 16592.251,E2 16592.251} C_VEL
LIN {X 0,Y 453.804,Z 1029.62,A -85,B 0,C 180,E1 16591.002,E2 16591.002} C_VEL
LIN {X 0,Y 460.826,Z 1008.548,A -85,B 0,C 180,E1 16589.778,E2 16589.778} C_VEL
LIN {X 0,Y 468.719,Z 981.603,A -85,B 0,C 180,E1 16588.485,E2 16588.485} C_VEL
LIN {X 0,Y 474.244,Z 959.484,A -85,B 0,C 180,E1 16587.614,E2 16587.614} C_VEL
LIN {X 0,Y 478.774,Z 938.464,A -85,B 0,C 180,E1 16586.929,E2 16586.929} C_VEL
LIN {X 0,Y 482.607,Z 917.148,A -85,B 0,C 180,E1 16586.356,E2 16586.356} C_VEL
LIN {X 0,Y 486.327,Z 891.134,A -85,B 0,C 180,E1 16585.809,E2 16585.809} C_VEL
LIN {X 0,Y 489.69,Z 851.605,A -85,B 0,C 180,E1 16585.166,E2 16585.166} C_VEL
LIN {X 0,Y 506.291,Z 632.395,A -85,B 0,C 180,E1 16581.765,E2 16581.765} C_VEL
LIN {X 0,Y 508.311,Z 605.938,A -85,B 0,C 180,E1 16581.341,E2 16581.341} C_VEL
LIN {X 0,Y 501.699,Z 595.445,A -85,B 0,C 180,E1 16578.837,E2 16578.837} C_VEL
LIN {X 0,Y 495.515,Z 586.148,A -85,B 0,C 180,E1 16576.109,E2 16576.109} C_VEL
LIN {X 0,Y 492.194,Z 581.305,A -85,B 0,C 180,E1 16574.41,E2 16574.41} C_VEL
LIN {X 0,Y 489.342,Z 577.099,A -85,B 0,C 180,E1 16572.749,E2 16572.749} C_VEL
LIN {X 0,Y 486.294,Z 572.605,A -85,B 0,C 180,E1 16570.664,E2 16570.664} C_VEL
LIN {X 0,Y 483.314,Z 568.269,A -85,B 0,C 180,E1 16568.087,E2 16568.087} C_VEL
LIN {X 0,Y 482.641,Z 567.344,A -85,B 0,C 180,E1 16567.38,E2 16567.38} C_VEL
LIN {X 0,Y 480.043,Z 563.601,A -85,B 0,C 180,E1 16563.344,E2 16563.344} C_VEL
LIN {X 0,Y 479.71,Z 561.956,A -85,B 0,C 180,E1 16561.792,E2 16561.792} C_VEL
LIN {X 0,Y 479.792,Z 562.179,A -85,B 0,C 180,E1 16558.209,E2 16558.209} C_VEL
LIN {X 0,Y 481.468,Z 566.289,A -85,B 0,C 180,E1 16554.399,E2 16554.399} C_VEL
LIN {X 0,Y 483.208,Z 568.007,A -85,B 0,C 180,E1 16552.45,E2 16552.45} C_VEL
LIN {X 0,Y 485.889,Z 572.231,A -85,B 0,C 180,E1 16550.046,E2 16550.046} C_VEL
LIN {X 0,Y 487.082,Z 573.772,A -85,B 0,C 180,E1 16549.174,E2 16549.174} C_VEL
LIN {X 0,Y 490.572,Z 578.915,A -85,B 0,C 180,E1 16546.924,E2 16546.924} C_VEL
LIN {X 0,Y 494.413,Z 584.575,A -85,B 0,C 180,E1 16544.847,E2 16544.847} C_VEL
LIN {X 0,Y 500.828,Z 595.619,A -85,B 0,C 180,E1 16541.871,E2 16541.871} C_VEL
LIN {X 0,Y 506.962,Z 606.636,A -85,B 0,C 180,E1 16539.447,E2 16539.447} C_VEL
LIN {X 0,Y 508.393,Z 609.519,A -85,B 0,C 180,E1 16538.916,E2 16538.916} C_VEL
LIN {X 0,Y 491.907,Z 826.669,A -85,B 0,C 180,E1 16535.543,E2 16535.543} C_VEL
LIN {X 0,Y 486.438,Z 897.81,A -85,B 0,C 180,E1 16534.417,E2 16534.417} C_VEL
LIN {X 0,Y 482.653,Z 926.946,A -85,B 0,C 180,E1 16533.859,E2 16533.859} C_VEL
LIN {X 0,Y 478.278,Z 951.023,A -85,B 0,C 180,E1 16533.268,E2 16533.268} C_VEL
LIN {X 0,Y 473.767,Z 971.78,A -85,B 0,C 180,E1 16532.635,E2 16532.635} C_VEL
LIN {X 0,Y 468.459,Z 992.95,A -85,B 0,C 180,E1 16531.855,E2 16531.855} C_VEL
LIN {X 0,Y 462.069,Z 1015.393,A -85,B 0,C 180,E1 16530.864,E2 16530.864} C_VEL
LIN {X 0,Y 453.451,Z 1041.833,A -85,B 0,C 180,E1 16529.443,E2 16529.443} C_VEL
LIN {X 0,Y 445.821,Z 1062.832,A -85,B 0,C 180,E1 16528.087,E2 16528.087} C_VEL
LIN {X 0,Y 438.81,Z 1080.706,A -85,B 0,C 180,E1 16526.753,E2 16526.753} C_VEL
LIN {X 0,Y 431.28,Z 1098.624,A -85,B 0,C 180,E1 16525.226,E2 16525.226} C_VEL
LIN {X 0,Y 422.039,Z 1119.436,A -85,B 0,C 180,E1 16523.173,E2 16523.173} C_VEL
LIN {X 0,Y 412.039,Z 1140.467,A -85,B 0,C 180,E1 16520.701,E2 16520.701} C_VEL
LIN {X 0,Y 404.241,Z 1156.233,A -85,B 0,C 180,E1 16518.55,E2 16518.55} C_VEL
LIN {X 0,Y 396.501,Z 1171.535,A -85,B 0,C 180,E1 16516.162,E2 16516.162} C_VEL
LIN {X 0,Y 389.002,Z 1186.184,A -85,B 0,C 180,E1 16513.543,E2 16513.543} C_VEL
LIN {X 0,Y 380.164,Z 1203.479,A -85,B 0,C 180,E1 16509.929,E2 16509.929} C_VEL
LIN {X 0,Y 373.477,Z 1216.671,A -85,B 0,C 180,E1 16506.663,E2 16506.663} C_VEL
LIN {X 0,Y 368.067,Z 1227.845,A -85,B 0,C 180,E1 16503.474,E2 16503.474} C_VEL
LIN {X 0,Y 363.55,Z 1237.744,A -85,B 0,C 180,E1 16500.226,E2 16500.226} C_VEL
LIN {X 0,Y 359.12,Z 1248.524,A -85,B 0,C 180,E1 16496.105,E2 16496.105} C_VEL
LIN {X 0,Y 355.803,Z 1257.681,A -85,B 0,C 180,E1 16491.781,E2 16491.781} C_VEL
LIN {X 0,Y 354.03,Z 1263.837,A -85,B 0,C 180,E1 16488.277,E2 16488.277} C_VEL
LIN {X 0,Y 352.902,Z 1268.671,A -85,B 0,C 180,E1 16484.945,E2 16484.945} C_VEL
LIN {X 0,Y 352.303,Z 1272.515,A -85,B 0,C 180,E1 16481.632,E2 16481.632} C_VEL
LIN {X 0,Y 352.021,Z 1275.396,A -85,B 0,C 180,E1 16478.336,E2 16478.336} C_VEL
LIN {X 0,Y 351.96,Z 1277.256,A -85,B 0,C 180,E1 16475.223,E2 16475.223} C_VEL
LIN {X 0,Y 351.958,Z 1278.269,A -85,B 0,C 180,E1 16472.124,E2 16472.124} C_VEL
LIN {X 0,Y 351.935,Z 1278.411,A -85,B 0,C 180,E1 16468.868,E2 16468.868} C_VEL
LIN {X 0,Y 351.957,Z 1277.615,A -85,B 0,C 180,E1 16465.608,E2 16465.608} C_VEL
LIN {X 0,Y 351.994,Z 1275.874,A -85,B 0,C 180,E1 16462.335,E2 16462.335} C_VEL
LIN {X 0,Y 352.248,Z 1273.021,A -85,B 0,C 180,E1 16458.879,E2 16458.879} C_VEL
LIN {X 0,Y 352.796,Z 1269.323,A -85,B 0,C 180,E1 16455.566,E2 16455.566} C_VEL
LIN {X 0,Y 353.82,Z 1264.641,A -85,B 0,C 180,E1 16452.238,E2 16452.238} C_VEL
LIN {X 0,Y 355.394,Z 1258.947,A -85,B 0,C 180,E1 16448.901,E2 16448.901} C_VEL
LIN {X 0,Y 357.687,Z 1252.21,A -85,B 0,C 180,E1 16445.571,E2 16445.571} C_VEL
LIN {X 0,Y 360.904,Z 1243.971,A -85,B 0,C 180,E1 16442.091,E2 16442.091} C_VEL
LIN {X 0,Y 365.914,Z 1232.596,A -85,B 0,C 180,E1 16437.997,E2 16437.997} C_VEL
LIN {X 0,Y 372.027,Z 1219.626,A -85,B 0,C 180,E1 16434.144,E2 16434.144} C_VEL
LIN {X 0,Y 378.092,Z 1207.386,A -85,B 0,C 180,E1 16431.005,E2 16431.005} C_VEL
LIN {X 0,Y 384.739,Z 1194.389,A -85,B 0,C 180,E1 16428.106,E2 16428.106} C_VEL
LIN {X 0,Y 393.477,Z 1177.554,A -85,B 0,C 180,E1 16424.861,E2 16424.861} C_VEL
LIN {X 0,Y 402.688,Z 1159.267,A -85,B 0,C 180,E1 16421.908,E2 16421.908} C_VEL
LIN {X 0,Y 410.289,Z 1143.931,A -85,B 0,C 180,E1 16419.76,E2 16419.76} C_VEL
LIN {X 0,Y 417.753,Z 1128.368,A -85,B 0,C 180,E1 16417.843,E2 16417.843} C_VEL
LIN {X 0,Y 425.929,Z 1110.607,A -85,B 0,C 180,E1 16415.929,E2 16415.929} C_VEL
LIN {X 0,Y 435.753,Z 1088.097,A -85,B 0,C 180,E1 16413.85,E2 16413.85} C_VEL
LIN {X 0,Y 444.523,Z 1066.004,A -85,B 0,C 180,E1 16412.142,E2 16412.142} C_VEL
LIN {X 0,Y 451.766,Z 1046.339,A -85,B 0,C 180,E1 16410.84,E2 16410.84} C_VEL
LIN {X 0,Y 458.255,Z 1027.149,A -85,B 0,C 180,E1 16409.742,E2 16409.742} C_VEL
LIN {X 0,Y 464.585,Z 1006.529,A -85,B 0,C 180,E1 16408.732,E2 16408.732} C_VEL
LIN {X 0,Y 471.769,Z 979.956,A -85,B 0,C 180,E1 16407.652,E2 16407.652} C_VEL
LIN {X 0,Y 477.311,Z 955.25,A -85,B 0,C 180,E1 16406.857,E2 16406.857} C_VEL
LIN {X 0,Y 481.376,Z 933.745,A -85,B 0,C 180,E1 16406.303,E2 16406.303} C_VEL
LIN {X 0,Y 484.748,Z 911.454,A -85,B 0,C 180,E1 16405.838,E2 16405.838} C_VEL
LIN {X 0,Y 487.612,Z 883.819,A -85,B 0,C 180,E1 16405.354,E2 16405.354} C_VEL
LIN {X 0,Y 503.976,Z 664.75,A -85,B 0,C 180,E1 16401.947,E2 16401.947} C_VEL
LIN {X 0,Y 508.243,Z 609.125,A -85,B 0,C 180,E1 16401.072,E2 16401.072} C_VEL
LIN {X 0,Y 501.18,Z 596.389,A -85,B 0,C 180,E1 16398.344,E2 16398.344} C_VEL
LIN {X 0,Y 495.527,Z 586.818,A -85,B 0,C 180,E1 16395.808,E2 16395.808} C_VEL
LIN {X 0,Y 492.545,Z 581.931,A -85,B 0,C 180,E1 16394.279,E2 16394.279} C_VEL
LIN {X 0,Y 488.971,Z 576.76,A -85,B 0,C 180,E1 16392.225,E2 16392.225} C_VEL
LIN {X 0,Y 486.165,Z 572.616,A -85,B 0,C 180,E1 16390.308,E2 16390.308} C_VEL
LIN {X 0,Y 483.265,Z 568.446,A -85,B 0,C 180,E1 16387.849,E2 16387.849} C_VEL
LIN {X 0,Y 482.584,Z 567.399,A -85,B 0,C 180,E1 16387.141,E2 16387.141} C_VEL
LIN {X 0,Y 479.955,Z 563.826,A -85,B 0,C 180,E1 16383.344,E2 16383.344} C_VEL
LIN {X 0,Y 479.51,Z 561.951,A -85,B 0,C 180,E1 16381.673,E2 16381.673} C_VEL
LIN {X 0,Y 479.62,Z 562.208,A -85,B 0,C 180,E1 16377.371,E2 16377.371} C_VEL
LIN {X 0,Y 480.965,Z 565.758,A -85,B 0,C 180,E1 16374.273,E2 16374.273} C_VEL
LIN {X 0,Y 483.021,Z 567.91,A -85,B 0,C 180,E1 16371.908,E2 16371.908} C_VEL
LIN {X 0,Y 485.812,Z 572.203,A -85,B 0,C 180,E1 16369.445,E2 16369.445} C_VEL
LIN {X 0,Y 486.93,Z 573.715,A -85,B 0,C 180,E1 16368.631,E2 16368.631} C_VEL
LIN {X 0,Y 490.545,Z 579.021,A -85,B 0,C 180,E1 16366.323,E2 16366.323} C_VEL
LIN {X 0,Y 494.271,Z 584.45,A -85,B 0,C 180,E1 16364.326,E2 16364.326} C_VEL
LIN {X 0,Y 499.426,Z 592.092,A -85,B 0,C 180,E1 16361.954,E2 16361.954} C_VEL
LIN {X 0,Y 506.004,Z 602.446,A -85,B 0,C 180,E1 16359.346,E2 16359.346} C_VEL
LIN {X 0,Y 508.207,Z 606.11,A -85,B 0,C 180,E1 16358.547,E2 16358.547} C_VEL
LIN {X 0,Y 491.848,Z 820.777,A -85,B 0,C 180,E1 16355.217,E2 16355.217} C_VEL
LIN {X 0,Y 486.893,Z 884.371,A -85,B 0,C 180,E1 16354.21,E2 16354.21} C_VEL
LIN {X 0,Y 483.03,Z 913.973,A -85,B 0,C 180,E1 16353.623,E2 16353.623} C_VEL
LIN {X 0,Y 478.955,Z 937.003,A -85,B 0,C 180,E1 16353.018,E2 16353.018} C_VEL
LIN {X 0,Y 474.563,Z 957.639,A -85,B 0,C 180,E1 16352.354,E2 16352.354} C_VEL
LIN {X 0,Y 469.526,Z 978.079,A -85,B 0,C 180,E1 16351.566,E2 16351.566} C_VEL
LIN {X 0,Y 463.258,Z 1000.369,A -85,B 0,C 180,E1 16350.547,E2 16350.547} C_VEL
LIN {X 0,Y 454.91,Z 1026.248,A -85,B 0,C 180,E1 16349.111,E2 16349.111} C_VEL
LIN {X 0,Y 447.704,Z 1046.059,A -85,B 0,C 180,E1 16347.811,E2 16347.811} C_VEL
LIN {X 0,Y 440.435,Z 1064.51,A -85,B 0,C 180,E1 16346.41,E2 16346.41} C_VEL
LIN {X 0,Y 432.852,Z 1082.462,A -85,B 0,C 180,E1 16344.844,E2 16344.844} C_VEL
LIN {X 0,Y 424.476,Z 1101.077,A -85,B 0,C 180,E1 16342.976,E2 16342.976} C_VEL
LIN {X 0,Y 413.866,Z 1123.049,A -85,B 0,C 180,E1 16340.37,E2 16340.37} C_VEL
LIN {X 0,Y 405.61,Z 1139.303,A -85,B 0,C 180,E1 16338.101,E2 16338.101} C_VEL
LIN {X 0,Y 398.322,Z 1153.25,A -85,B 0,C 180,E1 16335.871,E2 16335.871} C_VEL
LIN {X 0,Y 390.769,Z 1167.426,A -85,B 0,C 180,E1 16333.282,E2 16333.282} C_VEL
LIN {X 0,Y 382.137,Z 1183.525,A -85,B 0,C 180,E1 16329.859,E2 16329.859} C_VEL
LIN {X 0,Y 374.993,Z 1196.833,A -85,B 0,C 180,E1 16326.474,E2 16326.474} C_VEL
LIN {X 0,Y 369.423,Z 1207.54,A -85,B 0,C 180,E1 16323.318,E2 16323.318} C_VEL
LIN {X 0,Y 364.714,Z 1216.99,A -85,B 0,C 180,E1 16320.103,E2 16320.103} C_VEL
LIN {X 0,Y 360.383,Z 1226.455,A -85,B 0,C 180,E1 16316.34,E2 16316.34} C_VEL
LIN {X 0,Y 356.615,Z 1235.648,A -85,B 0,C 180,E1 16311.863,E2 16311.863} C_VEL
LIN {X 0,Y 354.559,Z 1241.699,A -85,B 0,C 180,E1 16308.233,E2 16308.233} C_VEL
LIN {X 0,Y 353.242,Z 1246.429,A -85,B 0,C 180,E1 16304.75,E2 16304.75} C_VEL
